// TwinCAT 3 PLC project CX_322E40
// libraries:
//   Tc2_ControllerToolbox, * (Beckhoff Automation GmbH)
//   Tc2_Coupler, * (Beckhoff Automation GmbH)
//   Tc2_DALI, * (Beckhoff Automation GmbH)
//   Tc2_EIB, * (Beckhoff Automation GmbH)
//   Tc2_EtherCAT, * (Beckhoff Automation GmbH)
//   Tc2_IoFunctions, * (Beckhoff Automation GmbH)
//   Tc2_LON, * (Beckhoff Automation GmbH)
//   Tc2_MBus, * (Beckhoff Automation GmbH)
//   Tc2_ModbusRTU, * (Beckhoff Automation GmbH)
//   Tc2_ModbusSrv, * (Beckhoff Automation GmbH)
//   Tc2_Standard, * (Beckhoff Automation GmbH)
//   Tc2_Standard, * (Beckhoff Automation GmbH)
//   Tc2_System, * (Beckhoff Automation GmbH)
//   Tc2_System, * (Beckhoff Automation GmbH)
//   Tc2_SystemCX, * (Beckhoff Automation GmbH)
//   Tc2_Utilities, * (Beckhoff Automation GmbH)
//   Tc3_Module, * (Beckhoff Automation GmbH)
//   Tc3_Module, * (Beckhoff Automation GmbH)
//   Tc3_PLCopen_OpcUa, * (Beckhoff Automation GmbH)
// project tree:
//   / ComTask.TcTTO, MBus_Zaehler_Task.TcTTO (not stored), Standard.TcTTO (not stored)
//   Data types/Anlagen/M2M/ WZM_EMAG_VLC100Y.TcDUT (not stored) (excluded from build)
//   Data types/Anlagen/ Machine2Machine.TcDUT (not stored)
//   Data types/Einzelanlagen/Absorptionskältemaschine %28AKM%29/ ST_AKM_Parameter.TcDUT (not stored), ST_AKM_Steuerung.TcDUT (not stored), ST_AKM_Zustand.TcDUT (not stored)
//   Data types/Einzelanlagen/Ampel/ ST_Ampel_Parameter.TcDUT (not stored), ST_Ampel_Steuerung.TcDUT, ST_Ampel_Zustand.TcDUT (not stored)
//   Data types/Einzelanlagen/Beleuchtung %28Bel%29/ ST_Bel_Lampen_Monitoring.TcDUT (not stored), ST_Bel_Parameter.TcDUT (not stored), ST_Bel_RGBW_Steuerung.TcDUT (not stored), ST_Bel_RGBW_Zustand.TcDUT (not stored), ST_Bel_Stellwert.TcDUT (not stored), ST_Bel_Steuerung.TcDUT (not stored), ST_Bel_Zustand.TcDUT (not stored)
//   Data types/Einzelanlagen/Betonspeicher %28BSp%29/ ST_BSp_Parameter.TcDUT (not stored), ST_Bsp_Steuerung.TcDUT (not stored), ST_BSp_Zustand.TcDUT (not stored)
//   Data types/Einzelanlagen/Blockheizkraftwerk %28BHKW%29/ ST_BHKW_Parameter.TcDUT (not stored), ST_BHKW_Stellwert.TcDUT (not stored), ST_BHKW_Steuerung.TcDUT (not stored), ST_BHKW_Zustand.TcDUT (not stored)
//   Data types/Einzelanlagen/Brennwertkessel %28BWK%29/ ST_BWK_Parameter.TcDUT (not stored), ST_BWK_Stellwert.TcDUT (not stored), ST_BWK_Steuerung.TcDUT (not stored), ST_BWK_Zustand.TcDUT (not stored)
//   Data types/Einzelanlagen/DC Schaltschrank %28DCSS%29/ ST_DCSS_Zustand.TcDUT (not stored)
//   Data types/Einzelanlagen/Druckluftkompressor %28DLK%29/ ST_DLK_Parameter.TcDUT (not stored), ST_DLK_Zustand.TcDUT (not stored)
//   Data types/Einzelanlagen/Drucksensor %28DS%29/ ST_DS_Parameter.TcDUT (not stored), ST_DS_Zustand.TcDUT (not stored)
//   Data types/Einzelanlagen/Fenster/ ST_Fenster_Parameter.TcDUT (not stored), ST_Fenster_Stellwert.TcDUT, ST_Fenster_Steuerung.TcDUT (not stored), ST_Fenster_Zustand.TcDUT (not stored)
//   Data types/Einzelanlagen/Gaszaehler %28GZ%29/ ST_GZ_DLK_Zustand.TcDUT (not stored), ST_GZ_Zustand.TcDUT (not stored)
//   Data types/Einzelanlagen/Haerteofen %28HO%29/ ST_HO_Parameter.TcDUT (not stored), ST_HO_Zustand.TcDUT (not stored)
//   Data types/Einzelanlagen/Heizstaebe %28HS%29/ ST_HS_Zustand.TcDUT (not stored)
//   Data types/Einzelanlagen/Hybrider Energiespeicher %28HES%29/ ST_HES_Parameter.TcDUT (not stored), ST_HES_Zustand.TcDUT (not stored)
//   Data types/Einzelanlagen/Kaeltekompressor %28KK%29/ ST_KKKW_Zustand.TcDUT (not stored)
//   Data types/Einzelanlagen/Lueftungsanlage %28LA%29/ ST_LA_Parameter.TcDUT (not stored), ST_LA_Stellwert.TcDUT (not stored), ST_LA_Steuerung.TcDUT (not stored), ST_LA_Zustand.TcDUT (not stored)
//   Data types/Einzelanlagen/Maschinenversorgung %28MV%29/ ST_MV_EMAG_VLC100Y_Zustand.TcDUT (not stored), ST_MV_HD_Zustand.TcDUT (not stored), ST_MV_JAVA_Parameter.TcDUT (not stored), ST_MV_JAVA_Zustand.TcDUT (not stored), ST_MV_MAFAC_GT_Parameter.TcDUT (not stored), ST_MV_MAFAC_GT_Zustand.TcDUT (not stored)
//   Data types/Einzelanlagen/Pufferspeicher %28PSp%29/ ST_PSp_Parameter.TcDUT (not stored), ST_PSp_Zustand.TcDUT (not stored)
//   Data types/Einzelanlagen/Pumpe %28Pu%29/ ST_PU_Genibus.TcDUT (not stored), ST_PU_Parameter.TcDUT (not stored), ST_PU_Stellwert.TcDUT (not stored), ST_PU_Steuerung.TcDUT (not stored), ST_PU_Zustand.TcDUT (not stored)
//   Data types/Einzelanlagen/Pumpe_lesend %28PU_Les%29/ ST_PU_les_Zustand.TcDUT (not stored)
//   Data types/Einzelanlagen/Pumpe_Schuetz %28PU_Schuetz%29/ ST_PU_Schuetz_Parameter.TcDUT (not stored), ST_PU_Schuetz_Stellwert.TcDUT (not stored), ST_PU_Schuetz_Steuerung.TcDUT (not stored), ST_PU_Schuetz_Zustand.TcDUT (not stored)
//   Data types/Einzelanlagen/Regelventil %28RV%29/ ST_RV_Parameter.TcDUT (not stored), ST_RV_Stellwert.TcDUT (not stored), ST_RV_Steuerung.TcDUT (not stored), ST_RV_Zustand.TcDUT (not stored)
//   Data types/Einzelanlagen/Regelventil_lesend %28RV_les%29/ ST_RV_les_Stellwert.TcDUT (not stored), ST_RV_les_Zustand.TcDUT (not stored)
//   Data types/Einzelanlagen/RGBW-Kanal/ ST_RGBW_Steuerung.TcDUT, ST_RGBW_Zustand.TcDUT (not stored)
//   Data types/Einzelanlagen/Signallampe GLT %28SL%29/ ST_SL_Parameter.TcDUT (not stored), ST_SL_Stellwert.TcDUT (not stored), ST_SL_Steuerung.TcDUT (not stored), ST_SL_Zustand.TcDUT (not stored)
//   Data types/Einzelanlagen/Stellventil %28SV%29 _ mit Status %28SVs%29/ ST_SVs_504_505_Zustand.TcDUT (not stored), ST_SVs_Zustand.TcDUT (not stored), ST_SV_Parameter.TcDUT (not stored), ST_SV_Stellwert.TcDUT (not stored), ST_SV_Steuerung.TcDUT (not stored), ST_SV_Zustand.TcDUT (not stored)
//   Data types/Einzelanlagen/Stromzaehler %28SZ%29/ ST_NSHV_Zustand.TcDUT (not stored), ST_SZ_Zustand.TcDUT (not stored)
//   Data types/Einzelanlagen/Tempfuehler%28TF%29/ ST_System_TF_Zustand.TcDUT (not stored)
//   Data types/Einzelanlagen/Waermepumpe %28WP%29/ ST_WP_Parameter.TcDUT (not stored), ST_WP_Stellwert.TcDUT (not stored), ST_WP_Steuerung.TcDUT (not stored), ST_WP_Zustand.TcDUT (not stored)
//   Data types/Einzelanlagen/Waermezaehler %28WZ%29/ ST_WZ_Zustand.TcDUT (not stored)
//   Data types/Library/Allgemein/ ST_Steuerung_auto_manu_BOOL.TcDUT (not stored), ST_Steuerung_auto_manu_opti_BOOL.TcDUT (not stored), ST_Steuerung_auto_manu_opti_REAL.TcDUT (not stored), ST_Steuerung_auto_manu_opti_SINT.TcDUT, ST_Steuerung_auto_manu_String.TcDUT, ST_Zustand_Netze_Anford.TcDUT (not stored), ST_Zustand_Netz_Anford.TcDUT (not stored)
//   Data types/Library/Bus_Systeme/ PB_64Byte.TcDUT (not stored), PB_Anfrage.TcDUT, PB_Dateneintrag.TcDUT, PB_GenibusType.TcDUT (not stored), PB_UMG604.TcDUT, ST_NSHV_Modbus.TcDUT
//   Data types/Management/ ST_FB_MGMT_Parameter.TcDUT (not stored), ST_FB_MGMT_Stellwert.TcDUT (not stored), ST_FB_MGMT_Steuerung.TcDUT, ST_FB_MGMT_Zustand.TcDUT (not stored), ST_MGMT_ThNTZ_Aktor_Parameter.TcDUT, ST_MGMT_ThNTZ_Aktor_Stellwert.TcDUT (not stored), ST_MGMT_ThNTZ_Aktor_Zustand.TcDUT (not stored)
//   Data types/Netze/ ST_Netze_Parameter.TcDUT (not stored), ST_Parameter_NTZ_Aktor_Regelung.TcDUT (not stored), ST_ThNTZ_Aktor.TcDUT, ST_ThNTZ_Parameter.TcDUT, ST_ThNTZ_Stellwert.TcDUT, ST_ThNTZ_Steuerung.TcDUT (not stored), ST_ThNTZ_Zustand.TcDUT
//   Data types/OPC-UA/ OPC_UA_BOOL.TcDUT (not stored), OPC_UA_REAL.TcDUT (not stored), ST_OPCUA_Node_BOOL.TcDUT, ST_OPCUA_Node_REAL.TcDUT (not stored), ST_OPCUA_Server.TcDUT, ST_OPC_UA_Node.TcDUT
//   Data types/Sonstige/ ST_GA_global.TcDUT (not stored), ST_Initialisierungsroutine.TcDUT (not stored)
//   Data types/Systeme/Anlagenversorgung %28AV%29/System Druckluftkompressor %28DLK%29/ ST_System_DLK_Parameter.TcDUT (not stored), ST_System_DLK_Stellwert.TcDUT (not stored), ST_System_DLK_Steuerung.TcDUT (not stored), ST_System_DLK_Zustand.TcDUT (not stored)
//   Data types/Systeme/Anlagenversorgung %28AV%29/System HybriderEnergiespeicher %28HES%29/ ST_System_HES_Parameter.TcDUT (not stored), ST_System_HES_Stellwert.TcDUT (not stored), ST_System_HES_Steuerung.TcDUT (not stored), ST_System_HES_Zustand.TcDUT (not stored)
//   Data types/Systeme/Anlagenversorgung %28AV%29/System Härteofen %28HO%29/System Härteofen Heisswasser %28HOHW%29/ ST_System_HOHW_Parameter.TcDUT (not stored), ST_System_HOHW_Stellwert.TcDUT (not stored), ST_System_HOHW_Steuerung.TcDUT (not stored), ST_System_HOHW_Zustand.TcDUT (not stored)
//   Data types/Systeme/Anlagenversorgung %28AV%29/System Härteofen %28HO%29/System Härteofen Warmwasser %28HOWW%29/ ST_System_HOWW_Parameter.TcDUT (not stored), ST_System_HOWW_Stellwert.TcDUT (not stored), ST_System_HOWW_Steuerung.TcDUT (not stored), ST_System_HOWW_Zustand.TcDUT (not stored)
//   Data types/Systeme/Anlagenversorgung %28AV%29/System Maschinenversorgung Heisswasser %28MVHW%29/ ST_System_MVHW_Parameter.TcDUT (not stored), ST_System_MVHW_Stellwert.TcDUT (not stored), ST_System_MVHW_Steuerung.TcDUT (not stored), ST_System_MVHW_Zustand.TcDUT (not stored)
//   Data types/Systeme/Anlagenversorgung %28AV%29/System Maschinenversorgung Kaltwasser %28MVKW%29/ ST_System_MVKW_Parameter.TcDUT (not stored), ST_System_MVKW_Stellwert.TcDUT (not stored), ST_System_MVKW_Steuerung.TcDUT (not stored), ST_System_MVKW_Zustand.TcDUT (not stored)
//   Data types/Systeme/Anlagenversorgung %28AV%29/System Maschinenversorgung Warmwasser %28MVWW%29/ ST_System_MVWW_Parameter.TcDUT (not stored), ST_System_MVWW_Stellwert.TcDUT (not stored), ST_System_MVWW_Steuerung.TcDUT (not stored), ST_System_MVWW_Zustand.TcDUT (not stored)
//   Data types/Systeme/Beleuchtung %28Bel%29/ ST_System_Bel_Parameter.TcDUT (not stored), ST_System_Bel_Stellwert.TcDUT (not stored), ST_System_Bel_Steuerung.TcDUT (not stored), ST_System_Bel_Zustand.TcDUT (not stored)
//   Data types/Systeme/Heizung_Klima_Lueftung/Klima/ ST_Klima_Aussen.TcDUT (not stored), ST_Klima_Bueros.TcDUT (not stored), ST_Klima_Halle.TcDUT
//   Data types/Systeme/Heizung_Klima_Lueftung/Lueftungsanlage %28LA%29/ ST_System_LA_Parameter.TcDUT (not stored), ST_System_LA_Stellwert.TcDUT (not stored), ST_System_LA_Steuerung.TcDUT (not stored), ST_System_LA_Zustand.TcDUT (not stored)
//   Data types/Systeme/Heizung_Klima_Lueftung/Lueftungsanlage %28LA%29/System_Fenster/ ST_System_Fenster_Parameter.TcDUT (not stored), ST_System_Fenster_Stellwert.TcDUT (not stored), ST_System_Fenster_Steuerung.TcDUT (not stored), ST_System_Fenster_Zustand.TcDUT (not stored)
//   Data types/Systeme/Heizung_Klima_Lueftung/Statische Heizung %28SHZ%29/ ST_System_SHZ_Parameter.TcDUT (not stored), ST_System_SHZ_Stellwert.TcDUT (not stored), ST_System_SHZ_Steuerung.TcDUT (not stored), ST_System_SHZ_Zustand.TcDUT (not stored)
//   Data types/Systeme/Heizung_Klima_Lueftung/ ST_Parameter_Kennlinie_Heizung_Kuehlung.TcDUT, ST_Parameter_Nachtabsenkung.TcDUT (not stored)
//   Data types/Systeme/Heizung_Klima_Lueftung/System Fussbodentemperierung %28FBT%29/ ST_System_FBT_Parameter.TcDUT (not stored), ST_System_FBT_Stellwert.TcDUT (not stored), ST_System_FBT_Steuerung.TcDUT (not stored), ST_System_FBT_Zustand.TcDUT (not stored)
//   Data types/Systeme/Heizung_Klima_Lueftung/Wand- & Deckentemperierung %28WDT%29/ ST_System_WDT_Parameter.TcDUT (not stored), ST_System_WDT_Stellwert.TcDUT (not stored), ST_System_WDT_Steuerung.TcDUT (not stored), ST_System_WDT_Zustand.TcDUT (not stored)
//   Data types/Systeme/Kaeltekompressor/Kaeltekompressor Kaltwasser/ ST_System_KKKW_Parameter.TcDUT, ST_System_KKKW_Stellwert.TcDUT, ST_System_KKKW_Steuerung.TcDUT (not stored), ST_System_KKKW_Zustand.TcDUT
//   Data types/Systeme/Speicher/Betonspeicher %28BSp%29/ ST_System_BSp_Parameter.TcDUT (not stored), ST_System_BSp_Stellwert.TcDUT (not stored), ST_System_BSp_Steuerung.TcDUT (not stored), ST_System_BSp_Zustand.TcDUT (not stored)
//   Data types/Systeme/Speicher/Betonspeicher Kühlwasser %28BSp_KueW%29/ ST_System_BSp_KueW_Parameter.TcDUT (not stored), ST_System_BSp_KueW_Stellwert.TcDUT (not stored), ST_System_BSp_KueW_Steuerung.TcDUT (not stored), ST_System_BSp_KueW_Zustand.TcDUT (not stored)
//   Data types/Systeme/Speicher/Betonspeicher Verbindung %28BSp_Verb%29/ ST_System_BSp_Verb_Parameter.TcDUT (not stored), ST_System_BSp_Verb_Stellwert.TcDUT (not stored), ST_System_BSp_Verb_Steuerung.TcDUT (not stored), ST_System_BSp_Verb_Zustand.TcDUT (not stored)
//   Data types/Systeme/System_Ampel/ ST_Steuerung_auto_manu_opti_AMPELSIGNAL.TcDUT, ST_System_Ampel_Signal.TcDUT, ST_System_Ampel_Stellwert.TcDUT, ST_System_Ampel_Steuerung.TcDUT (not stored), ST_System_Ampel_Zustand.TcDUT
//   Data types/Systeme/Wandler/Aussenfassadenaktivierung %28AFA%29/ ST_System_AFA_Parameter.TcDUT (not stored), ST_System_AFA_Stellwert.TcDUT (not stored), ST_System_AFA_Steuerung.TcDUT (not stored), ST_System_AFA_Zustand.TcDUT (not stored)
//   Data types/Systeme/Wandler/System Absorptionskältemaschine %28AKM%29/ ST_System_AKM_Parameter.TcDUT (not stored), ST_System_AKM_Stellwert.TcDUT (not stored), ST_System_AKM_Steuerung.TcDUT (not stored), ST_System_AKM_Zustand.TcDUT (not stored)
//   Data types/Systeme/Wandler/System Blockheizkraftwerk %28BHKW%29/ ST_System_BHKW_Parameter.TcDUT (not stored), ST_System_BHKW_Stellwert.TcDUT (not stored), ST_System_BHKW_Steuerung.TcDUT (not stored), ST_System_BHKW_Zustand.TcDUT (not stored)
//   Data types/Systeme/Wandler/System Brennwertkessel %28BWK%29/ ST_System_BWK_Parameter.TcDUT (not stored), ST_System_BWK_Stellwert.TcDUT (not stored), ST_System_BWK_Steuerung.TcDUT (not stored), ST_System_BWK_Zustand.TcDUT (not stored)
//   Data types/Systeme/Wandler/System Heizstaebe %28HS%29/ ST_System_HS_Parameter.TcDUT (not stored), ST_System_HS_Stellwert.TcDUT (not stored), ST_System_HS_Steuerung.TcDUT (not stored), ST_System_HS_Zustand.TcDUT (not stored)
//   Data types/Systeme/Wandler/System Waermepumpe %28WP%29/ ST_System_WP_Parameter.TcDUT (not stored), ST_System_WP_Stellwert.TcDUT (not stored), ST_System_WP_Steuerung.TcDUT (not stored), ST_System_WP_Zustand.TcDUT (not stored)
//   Data types/Systeme/Wandler/System Wärmetauscher Warm-Heisswasser %28WT_WHW%29/ ST_System_WT_HWW_Parameter.TcDUT (not stored), ST_System_WT_HWW_Stellwert.TcDUT (not stored), ST_System_WT_HWW_Steuerung.TcDUT (not stored), ST_System_WT_HWW_Zustand.TcDUT (not stored)
//   Global Variables/Anlagen Variablen/ Con_AFA.TcGVL, Con_AKM.TcGVL (not stored), Con_Bel.TcGVL (not stored), Con_BHKW.TcGVL, Con_BSp.TcGVL, Con_BWK.TcGVL (not stored), Con_DLK.TcGVL (not stored), Con_FBT.TcGVL (not stored), Con_HO.TcGVL, Con_HS.TcGVL (not stored), Con_KKKW.TcGVL, Con_MGMT.TcGVL (not stored), Con_MVKW.TcGVL (not stored), Con_MVWW.TcGVL, Con_PU.TcGVL, Con_RV.TcGVL (not stored), Con_SHZ.TcGVL, Con_SV.TcGVL, Con_ThNTZ.TcGVL, Con_WDT.TcGVL, Con_WP.TcGVL (not stored), Con_WT.TcGVL (not stored)
//   Global Variables/Bus_Systeme/ Modbus.TcGVL (not stored), M_Bus.TcGVL, Profibus.TcGVL
//   Global Variables/ Globale_Variablen.TcGVL (not stored), Global_Checks.TcGVL (not stored), Global_Variables.TcGVL, Variablen_Konfiguration.TcGVL (not stored)
//   POUs/Checks/ CheckBounds.TcPOU, CheckDivByte.TcPOU (not stored), CheckDivDint.TcPOU (not stored), CheckDivDWord.TcPOU, CheckDivInt.TcPOU (not stored), CheckDivLreal.TcPOU (not stored), CheckDivReal.TcPOU, CheckDivSInt.TcPOU (not stored), CheckDivWord.TcPOU, CheckRangeSigned.TcPOU (not stored), CheckRangeUnsigned.TcPOU
//   POUs/ com_task.TcPOU, Error_Catch.TcPOU, FB_GA_Allgemein.TcPOU (not stored), FB_Initialisierungsroutine.TcPOU, MAIN.TcPOU (not stored), MBUS_WZaehler.TcPOU, MBUS_Zaehler.TcPOU (not stored), P_EIB.TcPOU (excluded from build)
//   POUs/Einzelanlagen/Absorptionskältemaschine %28AKM%29/ FB_AKM.TcPOU (not stored), FB_AKM_Zuweisung.TcPOU (not stored)
//   POUs/Einzelanlagen/Ampel/ FB_Ampel.TcPOU (not stored), FB_Ampel_Out.TcPOU
//   POUs/Einzelanlagen/Beleuchtung %28Bel%29/Bel_RGBW/ FB_Bel_Einzel_farbe.TcPOU (not stored), FB_Bel_Einzel_farbe_1.TcPOU (not stored), FB_Bel_RGBW.TcPOU (not stored), FB_Bel_RGBW_Ablaufsteuerung.TcPOU (not stored), FB_Bel_RGBW_Logik.TcPOU (not stored), FB_Bel_RGBW_Regelung.TcPOU (not stored), FB_Bel_RGBW_Sued.TcPOU (not stored) (excluded from build)
//   POUs/Einzelanlagen/Beleuchtung %28Bel%29/ FB_Bel.TcPOU (not stored), FB_Bel_Ablaufsteuerung.TcPOU (not stored), FB_Bel_Filter.TcPOU (not stored), FB_Bel_Input.TcPOU (not stored), FB_Bel_Lichtsensor.TcPOU (not stored), FB_Bel_Logik.TcPOU (not stored), FB_Bel_Monitoring.TcPOU (not stored), FB_Bel_Output.TcPOU (not stored), FB_Bel_Sollwertscheck.TcPOU (not stored), FB_Bel_Stellwertscheck.TcPOU (not stored), FB_Bel_Steuerung.TcPOU (not stored), FB_Bel_Taster.TcPOU (not stored), FB_Bel_Taster_Steuerung.TcPOU (not stored), FB_Bel_Zustandscheck.TcPOU (not stored), F_Bel_Daten_Lesen.TcPOU (not stored), F_Bel_Daten_Schreiben.TcPOU (not stored)
//   POUs/Einzelanlagen/Betonspeicher %28BSp%29/ FB_BSp.TcPOU (not stored), FB_BSp_Input.TcPOU (not stored), FB_BSp_Zustandscheck.TcPOU (not stored)
//   POUs/Einzelanlagen/Blockheizkraftwerk %28BHKW%29/ FB_BHKW.TcPOU (not stored), FB_BHKW_Ablaufsteuerung.TcPOU (not stored), FB_BHKW_Input.TcPOU (not stored), FB_BHKW_Logik.TcPOU (not stored), FB_BHKW_Modbus.TcPOU (not stored), FB_BHKW_Output.TcPOU (not stored), FB_BHKW_Regelung.TcPOU (not stored), FB_BHKW_Sollwertscheck.TcPOU (not stored), FB_BHKW_Stellwertscheck.TcPOU (not stored), FB_BHKW_Zustandscheck.TcPOU (not stored), F_BHKW_Daten_Schreiben.TcPOU (not stored)
//   POUs/Einzelanlagen/Brennwertkessel %28BWK%29/ FB_BWK.TcPOU (not stored), FB_BWK_Ablaufsteuerung.TcPOU (not stored), FB_BWK_Input.TcPOU (not stored), FB_BWK_Logik.TcPOU (not stored), FB_BWK_Output.TcPOU (not stored), FB_BWK_Regelung.TcPOU (not stored), FB_BWK_SchreibeDaten.TcPOU (not stored), FB_BWK_Sollwertscheck.TcPOU (not stored), FB_BWK_Stellwertscheck.TcPOU (not stored), FB_BWK_Zustandscheck.TcPOU (not stored), LON_COM.TcPOU (not stored), LON_IN_OUT.TcPOU (not stored)
//   POUs/Einzelanlagen/DC Schaltschrank %28DCSS%29/ FB_DCSS.TcPOU (not stored)
//   POUs/Einzelanlagen/Druckluftkompressor %28DLK%29/ FB_DLK.TcPOU (not stored), FB_DLK_INIt.TcPOU (not stored), FB_DLK_Input.TcPOU (not stored), FB_DLK_Zustandscheck.TcPOU (not stored)
//   POUs/Einzelanlagen/Drucksensor/ FB_DS.TcPOU, FB_DS_Input.TcPOU, FB_DS_Zustandscheck.TcPOU
//   POUs/Einzelanlagen/Fenster/ FB_Fenster.TcPOU (not stored), FB_Fenster_Ablaufsteuerung.TcPOU (not stored), FB_Fenster_Logik.TcPOU, FB_Fenster_Output.TcPOU (not stored), FB_Fenster_Zustandscheck.TcPOU (not stored), F_Fenster_Daten_Lesen.TcPOU (not stored)
//   POUs/Einzelanlagen/Gaszähler/ FB_Gaszaehler.TcPOU (not stored), FB_GZ_DLK.TcPOU (not stored)
//   POUs/Einzelanlagen/Haerteofen %28HO%29/ FB_HO.TcPOU (not stored)
//   POUs/Einzelanlagen/Heizstab %28HS%29/ FB_HS.TcPOU (not stored)
//   POUs/Einzelanlagen/Hybrider Energiespeicher %28HES%29/ FB_HES.TcPOU (not stored)
//   POUs/Einzelanlagen/Kaeltekompressor %28KK%29/Kaeltekompressor Kaltwasser %28KKKW%29/ FB_KKKW.TcPOU (not stored)
//   POUs/Einzelanlagen/Lueftungsanlage %28LA%29/ FB_LA.TcPOU (not stored), FB_LA_Zustandscheck.TcPOU (not stored)
//   POUs/Einzelanlagen/Maschinenversorgung %28MV%29/ FB_MV_EMAG_GT.TcPOU (not stored), FB_MV_EMAG_VLC100Y.TcPOU (not stored), FB_MV_HD.TcPOU (not stored), FB_MV_JAVA.TcPOU (not stored)
//   POUs/Einzelanlagen/Pufferspeicher %28PSp%29/ FB_PSp.TcPOU (not stored), FB_PSp_Input.TcPOU (not stored), FB_PSp_Zustandscheck.TcPOU (not stored)
//   POUs/Einzelanlagen/Pumpe %28PU%29/ FB_PU.TcPOU (not stored), FB_PU_Ablaufsteuerung.TcPOU (not stored), FB_PU_Genibus.TcPOU (not stored), FB_PU_Genibus_old.TcPOU (not stored), FB_PU_Input.TcPOU (not stored), FB_PU_Logik.TcPOU (not stored), FB_PU_Output.TcPOU (not stored), FB_PU_Regelung.TcPOU (not stored), FB_PU_Sollwertscheck.TcPOU (not stored), FB_PU_Zustandscheck.TcPOU (not stored), F_PU_Daten_Schreiben.TcPOU (not stored)
//   POUs/Einzelanlagen/Pumpe %28PU%29/PU_191/ FB_PU_191.TcPOU (not stored), FB_PU_191_Ablaufsteuerung.TcPOU (not stored), FB_PU_191_Input.TcPOU (not stored)
//   POUs/Einzelanlagen/Pumpe Status %28PU_St%29/ FB_PU_St.TcPOU (not stored), FB_PU_St_Zustandscheck.TcPOU (not stored)
//   POUs/Einzelanlagen/Pumpe_lesend %28PU_les%29/ FB_PU_les.TcPOU (not stored), FB_PU_les_Genibus.TcPOU (not stored), FB_PU_les_Input.TcPOU (not stored)
//   POUs/Einzelanlagen/Pumpe_Schuetz %28PU_Schuetz%29/ FB_PU_Schuetz.TcPOU (not stored), FB_PU_Schuetz_Ablaufsteuerung.TcPOU (not stored), FB_PU_Schuetz_Logik.TcPOU (not stored), FB_PU_Schuetz_Output.TcPOU (not stored), FB_PU_Schuetz_Zustandscheck.TcPOU (not stored), FB_PU_Stellwertscheck.TcPOU (not stored)
//   POUs/Einzelanlagen/Regelventil %28RV%29/ FB_RV.TcPOU (not stored), FB_RV_Ablaufsteuerung.TcPOU (not stored), FB_RV_Logik.TcPOU (not stored), FB_RV_Output.TcPOU (not stored), FB_RV_Regelung.TcPOU (not stored), FB_RV_Sollwertscheck.TcPOU (not stored), FB_RV_Stellwertscheck.TcPOU (not stored), FB_RV_Zustandscheck.TcPOU (not stored)
//   POUs/Einzelanlagen/Regelventil Status %28RV_St%29/ FB_RV_St.TcPOU (not stored), FB_RV_St_Zustandscheck.TcPOU (not stored)
//   POUs/Einzelanlagen/Regelventil_lesend %28RV_les%29/ FB_RV_les.TcPOU (not stored)
//   POUs/Einzelanlagen/RGBW-Kanal/ FB_RGBW.TcPOU (not stored), FB_RGBW_Zustandscheck.TcPOU
//   POUs/Einzelanlagen/Stellventil %28SV%29/ FB_SV.TcPOU (not stored), FB_SV_Ablaufsteuerung.TcPOU (not stored), FB_SV_Logik.TcPOU (not stored), FB_SV_Output.TcPOU (not stored), FB_SV_Zustandscheck.TcPOU (not stored), F_SV_Daten_Schreiben.TcPOU (not stored)
//   POUs/Einzelanlagen/Stellventil mit Status %28SVs%29/ FB_SVs.TcPOU (not stored), FB_SVs_Ablaufsteuerung.TcPOU (not stored), FB_SVs_Input.TcPOU (not stored), FB_SVs_Logik.TcPOU (not stored), FB_SVs_Output.TcPOU (not stored), FB_SVs_Zustandscheck.TcPOU (not stored)
//   POUs/Einzelanlagen/Stellventil mit Status %28SVs%29/FB_SVs_504_505/ FB_SVs_504_505.TcPOU (not stored), FB_SVs_504_505_Ablaufsteuerung.TcPOU (not stored), FB_SVs_504_505_Input.TcPOU (not stored), FB_SVs_504_505_Logik.TcPOU (not stored), FB_SVs_504_505_Zustandscheck.TcPOU (not stored)
//   POUs/Einzelanlagen/Stromzähler/ABB_Stromzaehler/ FB_ABB_Lesen.TcPOU, FB_Stromzaehler.TcPOU (not stored), FB_Stromzaehler_BHKW.TcPOU, FB_Stromzaehler_Gebaeude.TcPOU
//   POUs/Einzelanlagen/Stromzähler/Netzanschlusspunkt/ FB_NSHV_Wert_zuweisen.TcPOU (not stored), FB_Stromzaehler_NSHV_Modbus.TcPOU
//   POUs/Einzelanlagen/Tempfuehler/ FB_TF.TcPOU (not stored)
//   POUs/Einzelanlagen/Waermepumpe/ FB_WP.TcPOU (not stored), FB_WP_Ablaufsteuerung.TcPOU, FB_WP_Logik.TcPOU, FB_WP_SchreibeDaten.TcPOU, FB_WP_Zustandscheck.TcPOU
//   POUs/Einzelanlagen/Wetterstation/ FB_WS.TcPOU (not stored), FB_WS_Init.TcPOU (not stored), FB_WS_Input.TcPOU (not stored), FB_WS_Konvertierung.TcPOU, FB_WS_Konvertierung_OLD.TcPOU (not stored), FB_WS_Mittelung.TcPOU
//   POUs/Einzelanlagen/Wärmezähler/ FB_Waermezaehler_MollineC3.TcPOU, FB_Waermezaehler_WP.TcPOU
//   POUs/Initialisierung/ P_init_dauernd.TcPOU (not stored), P_Init_einmalig.TcPOU (not stored)
//   POUs/Kommunikation/ FB_BUFFER_INT_TO_REAL.TcPOU, FB_BUFFER_REAL_TO_REAL.TcPOU, FB_BUFFER_UDINT_TO_REAL.TcPOU, OPC_UA_READ.TcPOU (not stored), OPC_UA_WRITE.TcPOU (not stored)
//   POUs/Library %28allgemein%29/ FB_SetResetFallTrigger.TcPOU (not stored), IEEE32_TO_REAL.TcPOU (not stored)
//   POUs/Management/Alte Struktur/ FB_MGMT_ThNTZ.TcPOU, FB_MGMT_ThNTZ_Aktor.TcPOU
//   POUs/Management/ FB_MGMT.TcPOU, FB_MGMT_Ablaufsteuerung.TcPOU, FB_MGMT_BSp.TcPOU (not stored), FB_MGMT_Logik.TcPOU, FB_MGMT_Regelung.TcPOU, FB_MGMT_Sollwertscheck.TcPOU, FB_MGMT_Zustandscheck.TcPOU (not stored), FB_Zuweisungen.TcPOU
//   POUs/OPC_UA_Client_Maschienen %28Romtech _ alt%29/ AKM_941_Read_BOOL.TcPOU (not stored) (excluded from build), AKM_941_Read_REAL.TcPOU (not stored) (excluded from build), AKM_941_Write_BOOL.TcPOU (not stored) (excluded from build), AKM_941_Write_REAL.TcPOU (not stored) (excluded from build), IVA_Ofen_Read_BOOL.TcPOU (not stored), IVA_Ofen_Read_REAL.TcPOU (not stored), PRG_Read_LREAL.TcPOU (not stored), SMS_Speicher_Read_BOOL.TcPOU (not stored) (excluded from build), SMS_Speicher_Read_REAL.TcPOU (not stored) (excluded from build)
//   POUs/Systeme/Anlagenversorgung %28AV%29/ FB_AV.TcPOU (not stored)
//   POUs/Systeme/Anlagenversorgung %28AV%29/Kühlung Druckluftkompressor %28DLK%29/ FB_System_DLK_951.TcPOU (not stored), FB_System_DLK_Ablaufsteuerung.TcPOU (not stored), FB_System_DLK_Logik.TcPOU (not stored), FB_System_DLK_Stellwertscheck.TcPOU (not stored), FB_System_DLK_Zustandscheck.TcPOU (not stored)
//   POUs/Systeme/Anlagenversorgung %28AV%29/Kühlung Hybrider Energiespeicher %28HES%29/ FB_System_HES_991.TcPOU (not stored), FB_System_HES_Ablaufsteuerung.TcPOU (not stored), FB_System_HES_Logik.TcPOU (not stored), FB_System_HES_Zustandscheck.TcPOU (not stored)
//   POUs/Systeme/Anlagenversorgung %28AV%29/Maschinenversorgung Heisswasser %28MVHW%29/ FB_System_MVHW_300.TcPOU (not stored), FB_System_MVHW_Ablaufsteuerung.TcPOU (not stored), FB_System_MVHW_Logik.TcPOU (not stored), FB_System_MVHW_Zustandscheck.TcPOU (not stored)
//   POUs/Systeme/Anlagenversorgung %28AV%29/Maschinenversorgung Kaltwasser %28MVKW%29/ FB_System_MVKW_100.TcPOU (not stored), FB_System_MVKW_Ablaufsteuerung.TcPOU (not stored), FB_System_MVKW_Logik.TcPOU (not stored), FB_System_MVKW_Zustandscheck.TcPOU (not stored)
//   POUs/Systeme/Anlagenversorgung %28AV%29/Maschinenversorgung Warmwasser %28MVWW%29/ FB_System_MVWW_245.TcPOU (not stored), FB_System_MVWW_Ablaufsteuerung.TcPOU (not stored), FB_System_MVWW_Logik.TcPOU (not stored), FB_System_MVWW_Sollwertscheck.TcPOU (not stored), FB_System_MVWW_Stellwertscheck.TcPOU (not stored), FB_System_MVWW_Zustandscheck.TcPOU (not stored)
//   POUs/Systeme/Anlagenversorgung %28AV%29/System Härteofen %28HO%29/ FB_System_HO_961.TcPOU (not stored)
//   POUs/Systeme/Anlagenversorgung %28AV%29/System Härteofen %28HO%29/System Härteofen Heisswasser %28HOHW%29/ FB_System_HOHW_361.TcPOU (not stored), FB_System_HOHW_Ablaufsteuerung.TcPOU (not stored), FB_System_HOHW_Logik.TcPOU (not stored), FB_System_HOHW_Zustandscheck.TcPOU (not stored)
//   POUs/Systeme/Anlagenversorgung %28AV%29/System Härteofen %28HO%29/System Härteofen Warmwasser %28HOWW%29/ FB_System_HOWW_261.TcPOU (not stored), FB_System_HOWW_Ablaufsteuerung.TcPOU (not stored), FB_System_HOWW_Logik.TcPOU (not stored), FB_System_HOWW_Zustandscheck.TcPOU (not stored)
//   POUs/Systeme/Heizung Lüftung Klimatisierung %28HLK%29/ FB_HLK.TcPOU (not stored)
//   POUs/Systeme/Heizung Lüftung Klimatisierung %28HLK%29/Fußbodentemperierung %28FBT%29/ FB_System_FBT_425.TcPOU (not stored), FB_System_FBT_Ablaufsteuerung.TcPOU (not stored), FB_System_FBT_Logik.TcPOU (not stored), FB_System_FBT_Regelung.TcPOU (not stored), FB_System_FBT_Sollwertscheck.TcPOU (not stored), FB_System_FBT_Stellwertscheck.TcPOU (not stored), FB_System_FBT_Zustandscheck.TcPOU (not stored)
//   POUs/Systeme/Heizung Lüftung Klimatisierung %28HLK%29/Raumlufttechnik %28RLT%29/Fenster %28FS%29/ FB_Fenster_Input.TcPOU (not stored), FB_System_Fenster.TcPOU (not stored), FB_System_Fenster_Logik.TcPOU (not stored), FB_System_Fenster_Regelung.TcPOU (not stored)
//   POUs/Systeme/Heizung Lüftung Klimatisierung %28HLK%29/Raumlufttechnik %28RLT%29/Lüftungsanlage %28LA%29/ FB_System_LA_955.TcPOU (not stored), FB_System_LA_Zustandscheck.TcPOU (not stored), SETINBYTE.TcPOU (not stored)
//   POUs/Systeme/Heizung Lüftung Klimatisierung %28HLK%29/Statische Heizung %28SHZ%29/ FB_System_SHZ_350.TcPOU (not stored), FB_System_SHZ_Ablaufsteuerung.TcPOU (not stored), FB_System_SHZ_Logik.TcPOU (not stored), FB_System_SHZ_Regelung.TcPOU (not stored), FB_System_SHZ_Sollwertscheck.TcPOU (not stored), FB_System_SHZ_Stellwertscheck.TcPOU (not stored), FB_System_SHZ_Zustandscheck.TcPOU (not stored)
//   POUs/Systeme/Heizung Lüftung Klimatisierung %28HLK%29/Wand- & Deckentemperierung %28WDT%29/ FB_System_WDT_500.TcPOU (not stored), FB_System_WDT_Ablaufsteuerung.TcPOU (not stored), FB_System_WDT_Logik.TcPOU (not stored), FB_System_WDT_Regelung.TcPOU (not stored), FB_System_WDT_Sollwertscheck.TcPOU (not stored), FB_System_WDT_Stellwertscheck.TcPOU (not stored), FB_System_WDT_Zustandscheck.TcPOU (not stored)
//   POUs/Systeme/Netze %28NTZ%29/ FB_HW_Zuweisungen.TcPOU (not stored), FB_KW_Zuweisungen.TcPOU (not stored), FB_NTZ.TcPOU (not stored), FB_NTZ_HW.TcPOU (not stored), FB_NTZ_KW.TcPOU (not stored), FB_NTZ_WW.TcPOU (not stored), FB_ThNTZ_Ablaufsteuerung.TcPOU (not stored), FB_ThNTZ_Logik.TcPOU (not stored), FB_ThNTZ_Regelung_Heissnetz.TcPOU (not stored), FB_ThNTZ_Regelung_Kaltnetz.TcPOU (not stored), FB_ThNTZ_Regelung_Warmnetz.TcPOU (not stored), FB_ThNTZ_Sollwertscheck.TcPOU (not stored), FB_ThNTZ_Zustandscheck.TcPOU (not stored), FB_WW_Zuweisungen.TcPOU (not stored)
//   POUs/Systeme/Sonstiges/Beleuchtung/Beleuchtung Außen/ FB_System_BelAu.TcPOU, FB_System_BelAu_Ablaufsteuerung.TcPOU, FB_System_BelAu_Logik.TcPOU, FB_System_BelAu_Regelung.TcPOU (not stored), FB_System_BelAu_Sensorik.TcPOU (not stored), FB_System_BelAu_Sollwertscheck.TcPOU, FB_System_BelAu_Stellwertscheck.TcPOU (not stored), FB_System_BelAu_Zustandscheck.TcPOU (not stored)
//   POUs/Systeme/Sonstiges/Beleuchtung/Beleuchtung Halle/ FB_System_BelHa.TcPOU (not stored), FB_System_BelHa_Ablaufsteuerung.TcPOU (not stored), FB_System_BelHa_Logik.TcPOU, FB_System_BelHa_Regelung.TcPOU (not stored), FB_System_BelHa_Sensorik.TcPOU (not stored), FB_System_BelHa_Sollwertscheck.TcPOU, FB_System_BelHa_Stellwertscheck.TcPOU (not stored), FB_System_BelHa_Zustandscheck.TcPOU (not stored)
//   POUs/Systeme/Sonstiges/Beleuchtung/ FB_Beleuchtung.TcPOU (not stored), FB_System_Bel_Zustandscheck.TcPOU
//   POUs/Systeme/Sonstiges/Signal_Ampel/ FB_System_Ampel.TcPOU (not stored), FB_System_Ampel_Sollwertscheck.TcPOU (not stored)
//   POUs/Systeme/Speicher %28SPR%29/Betonspeicher %28BSp%29/ FB_System_BSp_795.TcPOU (not stored), FB_System_BSp_795_Zustandscheck.TcPOU (not stored), FB_System_BSp_797.TcPOU (not stored), FB_System_BSp_797_Zustandscheck.TcPOU (not stored), FB_System_BSp_Ablaufsteuerung.TcPOU (not stored), FB_System_BSp_Logik.TcPOU (not stored), FB_System_BSp_Regelung.TcPOU (not stored), FB_System_BSp_Sollwertscheck.TcPOU (not stored), FB_System_BSp_Stellwertscheck.TcPOU (not stored)
//   POUs/Systeme/Speicher %28SPR%29/ FB_SPR.TcPOU (not stored)
//   POUs/Systeme/Wandler %28WDL%29/Absorptionskältemaschine %28AKM%29/ FB_System_AKM_941.TcPOU (not stored), FB_System_AKM_Ablaufsteuerung.TcPOU (not stored), FB_System_AKM_Logik.TcPOU (not stored), FB_System_AKM_Regelung.TcPOU (not stored), FB_System_AKM_Sollwertscheck.TcPOU (not stored), FB_System_AKM_Stellwertscheck.TcPOU (not stored), FB_System_AKM_Zustandscheck.TcPOU (not stored), FB_ThNTZ_Stellwertscheck.TcPOU (not stored)
//   POUs/Systeme/Wandler %28WDL%29/Aussenfassadenaktivierung %28AFA%29/ FB_System_AFA_600.TcPOU (not stored), FB_System_AFA_Ablaufsteuerung.TcPOU (not stored), FB_System_AFA_Logik.TcPOU (not stored), FB_System_AFA_Regelung.TcPOU (not stored), FB_System_AFA_Sollwertscheck.TcPOU (not stored), FB_System_AFA_Stellwertscheck.TcPOU (not stored), FB_System_AFA_Zustandscheck.TcPOU (not stored)
//   POUs/Systeme/Wandler %28WDL%29/Blockheizkraftwerke %28BHKWs%29/ FB_System_BHKW_921.TcPOU (not stored), FB_System_BHKW_922.TcPOU (not stored), FB_System_BHKW_Ablaufsteuerung.TcPOU (not stored), FB_System_BHKW_Logik.TcPOU (not stored), FB_System_BHKW_Sollwertscheck.TcPOU (not stored), FB_System_BHKW_Zustandscheck.TcPOU (not stored)
//   POUs/Systeme/Wandler %28WDL%29/Brennwertkessel %28BWK%29/ FB_System_BWK_931.TcPOU (not stored), FB_System_BWK_Ablaufsteuerung.TcPOU (not stored), FB_System_BWK_Logik.TcPOU (not stored), FB_System_BWK_Sollwertscheck.TcPOU (not stored), FB_System_BWK_Zustandscheck.TcPOU (not stored)
//   POUs/Systeme/Wandler %28WDL%29/ FB_WDL.TcPOU (not stored)
//   POUs/Systeme/Wandler %28WDL%29/Heizstaebe %28HS%29/ FB_System_HS_131.TcPOU (not stored), FB_System_HS_231.TcPOU (not stored), FB_System_HS_Logik.TcPOU (not stored), FB_System_HS_Regelung.TcPOU (not stored), FB_System_HS_Sollwertscheck.TcPOU (not stored), FB_System_HS_Zustandscheck.TcPOU (not stored)
//   POUs/Systeme/Wandler %28WDL%29/System_Kaeltekompressoren %28KK%29/Kältekompressor Kaltwasser/ FB_System_KKKW_145.TcPOU (not stored), FB_System_KKKW_Ablaufsteuerung.TcPOU (not stored), FB_System_KKKW_Logik.TcPOU (not stored), FB_System_KKKW_Sollwertscheck.TcPOU (not stored), FB_System_KKKW_Stellwertscheck.TcPOU (not stored), FB_System_KKKW_Zustandscheck.TcPOU (not stored)
//   POUs/Systeme/Wandler %28WDL%29/Waermepumpe %28WP%29/ FB_System_WP_946.TcPOU (not stored), FB_System_WP_Ablaufsteuerung.TcPOU (not stored), FB_System_WP_Logik.TcPOU (not stored), FB_System_WP_Zustandscheck.TcPOU (not stored)
//   POUs/Systeme/Wandler %28WDL%29/Wärmetauscher %28WT%29/ FB_System_WT_HWW_915.TcPOU (not stored), FB_System_WT_HWW_Ablaufsteuerung.TcPOU (not stored), FB_System_WT_HWW_Logik.TcPOU (not stored), FB_System_WT_HWW_Sollwertscheck.TcPOU (not stored), FB_System_WT_HWW_Zustandscheck.TcPOU (not stored)
//   POUs/Systeme/Zaehler %28ZAE%29/ FB_ZAE.TcPOU (not stored)
//   POUs/Umwelt/ FB_UMWELT.TcPOU, FB_UWT.TcPOU (not stored), FB_UW_Temp_Mittelung.TcPOU (not stored)

CONFIGURATION CX_322E40
    RESOURCE PLC ON TwinCAT3
        TASK ComTask(INTERVAL := T#25000us, PRIORITY := 6);
        PROGRAM com_task WITH ComTask : com_task;
    END_RESOURCE
END_CONFIGURATION

// ---- Data types/Einzelanlagen/Ampel/ST_Ampel_Steuerung.TcDUT
TYPE ST_Ampel_Steuerung :
STRUCT
	Freigabe			: ST_Steuerung_auto_manu_BOOL;
	Quittierung			: BOOL;
END_STRUCT
END_TYPE

// ---- Data types/Einzelanlagen/Fenster/ST_Fenster_Stellwert.TcDUT
TYPE ST_Fenster_Stellwert :
STRUCT
	Freigabe		: BOOL;
	Stellung		: BOOL;

	Fenster_AUF		: BOOL;
	Fenster_ZU		: BOOL;




END_STRUCT
END_TYPE

// ---- Data types/Einzelanlagen/RGBW-Kanal/ST_RGBW_Steuerung.TcDUT
TYPE ST_RGBW_Steuerung :
STRUCT
	Betrieb			: BOOL;
	Farbcode	: STRING;
END_STRUCT
END_TYPE

// ---- Data types/Library/Allgemein/ST_Steuerung_auto_manu_opti_SINT.TcDUT
TYPE ST_Steuerung_auto_manu_opti_SINT :
STRUCT
	auto			: SINT;
	manu			: SINT;
	manu_Modus		: BOOL;
	opti			: SINT;
	opti_Modus		: BOOL;
END_STRUCT
END_TYPE

// ---- Data types/Library/Allgemein/ST_Steuerung_auto_manu_String.TcDUT
TYPE ST_Steuerung_auto_manu_String :
STRUCT
	auto			: STRING;
	manu			: STRING;
	manu_Modus		: BOOL;
END_STRUCT
END_TYPE

// ---- Data types/Library/Bus_Systeme/PB_Anfrage.TcDUT
TYPE PB_Anfrage :
STRUCT
	pAuslass 			: PB_Dateneintrag;

	tAuslass 				: PB_Dateneintrag;
	
	tDruckTau			: PB_Dateneintrag;
	
	tUmgebung			: PB_Dateneintrag;

	tAqEin				: PB_Dateneintrag;

	tAqAus				: PB_Dateneintrag;
	
	mechState			: PB_Dateneintrag;

	hBetrieb				: PB_Dateneintrag;

	hGeringeLast			: PB_Dateneintrag;

	vErzeugtesVolumen	: PB_Dateneintrag;
END_STRUCT
END_TYPE

// ---- Data types/Library/Bus_Systeme/PB_Dateneintrag.TcDUT
TYPE PB_Dateneintrag :
STRUCT
	CANAdress 	: BYTE;
	Parameter 	: UINT;	
	Value		: UINT;
	Status		: WORD;
END_STRUCT
END_TYPE

// ---- Data types/Library/Bus_Systeme/PB_UMG604.TcDUT
TYPE PB_UMG604 :
(*Struktur für das Universalmessgerät 604 (Janitza) *)
STRUCT
	ProfilNummer		: BYTE;
	Wirkleistung 		: REAL;
	Blindleistung		: REAL;
	Scheinleistung	: REAL;
	Wirkarbeit		: REAL;
	Blindarbeit		: REAL;
	Scheinarbeit		: REAL;
	DiZaehlstand		: REAL;
	DiZustand		: REAL;
	DiLeistungswert	: REAL;
	NichtBelegt1		: REAL;
	NichtBelegt2		: REAL;
	NichtBelegt3		: REAL;
	NichtBelegt4		: REAL;
	NichtBelegt5		: REAL;
	NichtBelegt6		: REAL;
	NichtBelegt7		: REAL;
	NichtBelegt8		: REAL;
	NichtBelegt9		: REAL;
	NichtBelegt10		: REAL;
	NichtBelegt11		: REAL;
	NichtBelegt12		: REAL;
	NichtBelegt13		: REAL;
	NichtBelegt14		: REAL;
	NichtBelegt15		: REAL;
	NichtBelegt16		: REAL;
	NichtBelegt17		: REAL;
	NichtBelegt18		: REAL;
	NichtBelegt19		: REAL;
	NichtBelegt20		: REAL;
	NichtBelegt21		: REAL;
	NichtBelegt22		: REAL;
END_STRUCT
END_TYPE

// ---- Data types/Library/Bus_Systeme/ST_NSHV_Modbus.TcDUT
TYPE ST_NSHV_Modbus :
STRUCT
	Modbus_Unit_Online	: BOOL; (*True = online, False = Offline*)
	Modbus_Adresse1  : ARRAY[16#1000..16#1568] OF DWORD;
END_STRUCT
END_TYPE

// ---- Data types/Management/ST_FB_MGMT_Steuerung.TcDUT
TYPE ST_FB_MGMT_Steuerung :
STRUCT
	Freigabe			         : ST_Steuerung_auto_manu_BOOL;
	Freigabe_Deakt		: ST_Steuerung_auto_manu_BOOL;
	Betrieb_Anford		: ST_Steuerung_auto_manu_opti_BOOL;

	Regelung_Modus		: ST_Steuerung_auto_manu_opti_SINT;
	Regelung_Sollw		: ST_Steuerung_auto_manu_opti_REAL;
	Regelung_Sollw_Max	: ST_Steuerung_auto_manu_opti_REAL;
	Regelung_Sollw_Min	: ST_Steuerung_auto_manu_opti_REAL;

	Quittierung			: BOOL;

END_STRUCT
END_TYPE

// ---- Data types/Management/ST_MGMT_ThNTZ_Aktor_Parameter.TcDUT
TYPE ST_MGMT_ThNTZ_Aktor_Parameter :
STRUCT
	Anford_Netz_KW			: ST_Zustand_Netz_Anford;
	Anford_Netz_WW			: ST_Zustand_Netz_Anford;
	Anford_Netz_HW			: ST_Zustand_Netz_Anford;
	Regelung_Netz_KW		: ST_Parameter_NTZ_Aktor_Regelung;	(* Aktiv: Bool, Grenzwert_Oben: REAL, Grenzwert_Unten: REAL, Prioritaet: SINT;*)
	Regelung_Netz_WW		: ST_Parameter_NTZ_Aktor_Regelung;
	Regelung_Netz_HW		: ST_Parameter_NTZ_Aktor_Regelung;

	Kennlinie_Tctr			: DINT := 5000;
END_STRUCT
END_TYPE

// ---- Data types/Netze/ST_ThNTZ_Aktor.TcDUT
TYPE ST_ThNTZ_Aktor :
STRUCT
	Verfuegbarkeit_Heizer		: BOOL;
	Verfuegbarkeit_Kuehler	: BOOL;
	Betrieb_Heizer_Anford		: BOOL;
	Betrieb_Kuehler_Anford	: BOOL;
END_STRUCT
END_TYPE

// ---- Data types/Netze/ST_ThNTZ_Parameter.TcDUT
TYPE ST_ThNTZ_Parameter :
STRUCT
	Temp_Max				: REAL;
	Temp_Min				: REAL;
	Regelung_PI_Oben_Kp	: REAL;
	Regelung_PI_Oben_Tn	: DINT;
	Regelung_PI_Oben_Tctr	: DINT;

	Regelung_Sollw_KRITIKAL_OBEN_TEMP    : REAL;
	Regelung_Sollw_KRITIKAL_UNTEN_TEMP   : REAL;
	Regelung_Sollw_Max    : REAL;
	Regelung_Sollw_Min    : REAL;
	Regelung_Sollw_Max_Min : REAL;


	Stellwert_Leistung_Max		: REAL;
	Stellwert_Leistung_Min		: REAL;

	AutoQuittierung			: BOOL;



END_STRUCT
END_TYPE

// ---- Data types/Netze/ST_ThNTZ_Stellwert.TcDUT
TYPE ST_ThNTZ_Stellwert :
STRUCT
	Betrieb		: BOOL;
	Leistung	: REAL;
END_STRUCT
END_TYPE

// ---- Data types/Netze/ST_ThNTZ_Zustand.TcDUT
TYPE ST_ThNTZ_Zustand :
STRUCT
	Betrieb_Anford			: BOOL;
	Betrieb_Soll			: BOOL;
	Betrieb					: BOOL;

	Regelung_Modus				: SINT;
	Regelung_Sollw_Widerspruch	: BOOL;
	Regelung_Sollw				: REAL;
	Regelung_Sollw_Max          : REAL;
	Regelung_Sollw_Min			: REAL;

	Regelung_Sollw_Anford		: REAL;
	Regelung_Sollw_Oben			: REAL;
	Regelung_Sollw_Oben_Max		: REAL;
	Regelung_Sollw_Oben_Min		: REAL;
	Regelung_Sollw_Unten		: REAL;
	Regelung_Sollw_Unten_Max	: REAL;
	Regelung_Sollw_Unten_Min	: REAL;
	Regelung_Stellw				: REAL;
	Regelung_Istw				: REAL;

	Temp_Max				: REAL;
	Temp_Oben				: REAL;
	Temp_Min				: REAL;
	Temp_Unten				: REAL;

	Freigabe				: BOOL;
	Freigabe_Deakt			: BOOL;
	Freigabe_Code			: WORD;

    Netze_Anford            : ARRAY [1..20] OF ST_Zustand_Netze_Anford;

	Stoerung				: BOOL;
	Stoerung_Code			: WORD;

	Warnung					: BOOL;
	Warnung_Code			: WORD;

	Status					: SINT;

	Quittierung				: BOOL;

END_STRUCT
END_TYPE

// ---- Data types/OPC-UA/ST_OPCUA_Node_BOOL.TcDUT
TYPE ST_OPCUA_Node_BOOL :
STRUCT
	NodeID				: ST_UANodeID;
	NodeHdl				: DWORD;
	SizeOfDataType		: UDINT;
	NodeAddInfo			: ST_UANodeAdditionalInfo;
	TargetVar			: POINTER TO BOOL;
END_STRUCT
END_TYPE

// ---- Data types/OPC-UA/ST_OPCUA_Server.TcDUT
TYPE ST_OPCUA_Server :
STRUCT
	sServerURL				: STRING;
	SessionConnectInfo		: ST_UASessionConnectInfo := (	tConnectTimeout			:= T#5S,
															tSessionTimeout 		:= T#1M,
															sApplicationName		:= '',
															eSecurityMode 			:= eUASecurityMsgMode_None,
															eSecurityPolicyUri	 	:= eUASecurityPolicy_None,
															eTransportProfileUri 	:= eUATransportProfileUri_UATcp);
	tTimeout            	: TIME := T#5M;
	nConnectionHdl			: DWORD;
END_STRUCT
END_TYPE

// ---- Data types/OPC-UA/ST_OPC_UA_Node.TcDUT
TYPE ST_OPC_UA_Node :
STRUCT
	NodeID				: ST_UANodeID;
	NodeHdl				: DWORD;
	SizeOfDataType		: UDINT;
	NodeAddInfo			: ST_UANodeAdditionalInfo;
	TargetVar			: POINTER TO BOOL;
END_STRUCT
END_TYPE

// ---- Data types/Systeme/Heizung_Klima_Lueftung/Klima/ST_Klima_Halle.TcDUT
TYPE ST_Klima_Halle :
STRUCT
	Temperatur_Sektor1	: REAL;
	Temperatur_Sektor2	: REAL;
	Temperatur_Sektor3	: REAL;
END_STRUCT
END_TYPE

// ---- Data types/Systeme/Heizung_Klima_Lueftung/ST_Parameter_Kennlinie_Heizung_Kuehlung.TcDUT
TYPE ST_Parameter_Kennlinie_Heizung_Kuehlung :
STRUCT
	Temp_Vorl_Max			: REAL;
	Temp_Vorl_Min			: REAL;
	Temp_Aussen_Max			: REAL;
	Temp_Aussen_Min			: REAL;



END_STRUCT
END_TYPE

// ---- Data types/Systeme/Kaeltekompressor/Kaeltekompressor Kaltwasser/ST_System_KKKW_Parameter.TcDUT
TYPE ST_System_KKKW_Parameter :
STRUCT
		AutoQuittierung			: BOOL;
END_STRUCT
END_TYPE

// ---- Data types/Systeme/Kaeltekompressor/Kaeltekompressor Kaltwasser/ST_System_KKKW_Stellwert.TcDUT
TYPE ST_System_KKKW_Stellwert :
STRUCT
	Anford_Stellventil		: BOOL;
	Anford_Pumpe			: BOOL;
	Einschaltperiode_Max	: TIME := T#5S;
	Einschalten				: BOOL;
	Modus_Pumpe				: SINT;
	Sollw_Pumpe				: REAL;
END_STRUCT
END_TYPE

// ---- Data types/Systeme/Kaeltekompressor/Kaeltekompressor Kaltwasser/ST_System_KKKW_Zustand.TcDUT
TYPE ST_System_KKKW_Zustand :
STRUCT
	Betrieb_Anford			: BOOL;
	Betrieb_Soll				: BOOL;
	Betrieb					: BOOL;

	Regelung_Sollw			: REAL;
	Regelung_Modus				: SINT;

	Freigabe					: BOOL;
	Freigabe_Deakt			: BOOL;
	Freigabe_Code			: WORD;

	Stoerung					: BOOL;
	Stoerung_Code			: WORD;

	Warnung					: BOOL;
	Warnung_Code			: WORD;

	Status					: SINT;
	Status_Vorl				: BOOL;
	Status_Nachl				: BOOL;

	Status_Vorl_Stellventil	: BOOL;
	Status_Vorl_Pumpen		: BOOL;
	Status_Nachl_Stellventil: BOOL;
	Status_Nachl_Pumpen		: BOOL;
	Status_Wiedereinschalten: BOOL;

	Quittierung				: BOOL;

END_STRUCT
END_TYPE

// ---- Data types/Systeme/System_Ampel/ST_Steuerung_auto_manu_opti_AMPELSIGNAL.TcDUT
TYPE ST_Steuerung_auto_manu_opti_AMPELSIGNAL :
STRUCT
	auto			: ST_System_Ampel_Signal;
	manu			: ST_System_Ampel_Signal;
	manu_Modus		: BOOL;
	opti			: ST_System_Ampel_Signal;
	opti_Modus		: BOOL;
END_STRUCT
END_TYPE

// ---- Data types/Systeme/System_Ampel/ST_System_Ampel_Signal.TcDUT
TYPE ST_System_Ampel_Signal :
STRUCT
	Stellung_Rot		: BOOL;
	Stellung_Orange		: BOOL;
	Stellung_Gruen		: BOOL;
	Stellung_Blau		: BOOL;
	Stellung_Buzz		: BOOL;
END_STRUCT
END_TYPE

// ---- Data types/Systeme/System_Ampel/ST_System_Ampel_Stellwert.TcDUT
TYPE ST_System_Ampel_Stellwert :
STRUCT
	Stellung_Rot		: BOOL;
	Stellung_Orange		: BOOL;
	Stellung_Gruen		: BOOL;
	Stellung_Blau		: BOOL;
	Stellung_Buzz		: BOOL;
END_STRUCT
END_TYPE

// ---- Data types/Systeme/System_Ampel/ST_System_Ampel_Zustand.TcDUT
TYPE ST_System_Ampel_Zustand :
STRUCT
	Regelung_Sollw			: ST_System_Ampel_Signal;

	In_Ordnung			: BOOL;

	Stellung : ST_System_Ampel_Signal;
END_STRUCT
END_TYPE

// ---- Global Variables/Anlagen Variablen/Con_AFA.TcGVL
{attribute 'Tc2GvlVarNames'}
VAR_GLOBAL CONSTANT
	(* System_AFA_Zustand_Status *)
	E_System_AFA_Zustand_Status_Idle_Sperre			: SINT := 0;
	E_System_AFA_Zustand_Status_Betriebsbereit		: SINT := 1;
	E_System_AFA_Zustand_Status_Nachl_Pumpe			: SINT := 2;
	E_System_AFA_Zustand_Status_Vorl_Pumpe			: SINT := 3;
	E_System_AFA_Zustand_Status_Nachl_Regelventil	: SINT := 4;
	E_System_AFA_Zustand_Status_Vorl_Regelventil	: SINT := 5;
	E_System_AFA_Zustand_Status_Betrieb				: SINT := 6;
	E_System_AFA_Zustand_Status_Betrieb_Sperre		: SINT := 7;
	E_System_AFA_Zustand_Status_Stoerung			: SINT := 99;

	(* System_AFA_Zustand_Regelung_Modus *)
	E_System_AFA_Regelung_Modus_Wanddeckentemperierung		: SINT := -4;
	E_System_AFA_Regelung_Modus_Netz						: SINT := -5;

	E_System_AFA_Regelung_Modus_Waermeabsorber_Automatik	: SINT := 1;
	E_System_AFA_Regelung_Modus_Waermeabsorber_DachWaende	: SINT := 2;
	E_System_AFA_Regelung_Modus_Waermeabsorber_Dach			: SINT := 3;
	E_System_AFA_Regelung_Modus_Rueckkuehler_Automatik		: SINT := -1;
	E_System_AFA_Regelung_Modus_Rueckkuehler_DachWaende		: SINT := -2;
	E_System_AFA_Regelung_Modus_Rueckkuehler_Dach			: SINT := -3;

END_VAR

// ---- Global Variables/Anlagen Variablen/Con_BHKW.TcGVL
{attribute 'Tc2GvlVarNames'}
VAR_GLOBAL CONSTANT
	(* BHKW_Zustand_Status *)
	E_BHKW_Zustand_Status_Idle_Sperre			: SINT := 0;
	E_BHKW_Zustand_Status_Betriebsbereit		: SINT := 1;
	E_BHKW_Zustand_Status_Nachl					: SINT := 2;
	E_BHKW_Zustand_Status_Vorl					: SINT := 3;
	E_BHKW_Zustand_Status_Betrieb				: SINT := 4;
	E_BHKW_Zustand_Status_Betrieb_Sperre		: SINT := 5;
	E_BHKW_Zustand_Status_Stoerung				: SINT := 99;

	(* BHKW_Zustand_Regelung_Modus *)
	E_BHKW_Regelung_Modus_P						: SINT := 0;
	E_BHKW_Regelung_Modus_T_SH_Max				: SINT := 1;

	(* System_BHKW_Zustand_Status *)
	E_System_BHKW_Zustand_Status_Idle_Sperre		: SINT := 0;
	E_System_BHKW_Zustand_Status_Betriebsbereit		: SINT := 1;
	E_System_BHKW_Zustand_Status_Nachl_Stellventil	: SINT := 2;
	E_System_BHKW_Zustand_Status_Vorl_Stellventil	: SINT := 3;
	E_System_BHKW_Zustand_Status_Nachl_Pumpe		: SINT := 4;
	E_System_BHKW_Zustand_Status_Vorl_Pumpe			: SINT := 5;
	E_System_BHKW_Zustand_Status_Nachl_BHKW			: SINT := 6;
	E_System_BHKW_Zustand_Status_Vorl_BHKW			: SINT := 7;
	E_System_BHKW_Zustand_Status_Betrieb			: SINT := 8;
	E_System_BHKW_Zustand_Status_Betrieb_Sperre		: SINT := 9;
	E_System_BHKW_Zustand_Status_Ueberhitzt			: SINT := 10;
	E_System_BHKW_Zustand_Status_Stoerung			: SINT := 99;
END_VAR

// ---- Global Variables/Anlagen Variablen/Con_BSp.TcGVL
{attribute 'Tc2GvlVarNames'}
VAR_GLOBAL CONSTANT
	(* BSp_Zustand_Regelung_Modus *)
	E_BSp_Regelung_Modus_konst						: SINT := 0;
	E_BSp_Regelung_Modus_Laden_T_int				: SINT := 1;
	E_BSp_Regelung_Modus_Laden_T_ext				: SINT := 2;
	E_BSp_Regelung_Modus_Laden_dT					: SINT := 3;
	E_BSp_Regelung_Modus_Entladen_dT				: SINT := -3;
	E_BSp_Regelung_Modus_Entladen_T_int				: SINT := -1;
	E_BSp_Regelung_Modus_Entladen_T_ext				: SINT := -2;


	(* System_BSp_Zustand_Status *)
	E_System_BSp_Zustand_Status_Idle_Sperre			: SINT := 0;
	E_System_BSp_Zustand_Status_Betriebsbereit		: SINT := 1;
	E_System_BSp_Zustand_Status_Nachl_Stellventil	: SINT := 2;
	E_System_BSp_Zustand_Status_Vorl_Stellventil	: SINT := 3;
	E_System_BSp_Zustand_Status_Nachl_Pumpen		: SINT := 4;
	E_System_BSp_Zustand_Status_Vorl_Pumpen			: SINT := 5;
	E_System_BSp_Zustand_Status_Betrieb				: SINT := 8;
	E_System_BSp_Zustand_Status_Betrieb_Sperre		: SINT := 9;
	E_System_BSp_Zustand_Status_Stoerung			: SINT := 99;

	(* System_BSp_KueW_Zustand_Status *)
	E_System_BSp_KueW_Zustand_Status_Idle_Sperre	: SINT := 0;
	E_System_BSp_KueW_Zustand_Status_Betriebsbereit	: SINT := 1;
	E_System_BSp_KueW_Zustand_Status_Nachl			: SINT := 4;
	E_System_BSp_KueW_Zustand_Status_Vorl			: SINT := 5;
	E_System_BSp_KueW_Zustand_Status_Betrieb		: SINT := 8;
	E_System_BSp_KueW_Zustand_Status_Betrieb_Sperre	: SINT := 9;
	E_System_BSp_KueW_Zustand_Status_Stoerung		: SINT := 99;

	(* System_BSp_Verb_Zustand_Status *)
	E_System_BSp_Verb_Zustand_Status_Idle_Sperre	: SINT := 0;
	E_System_BSp_Verb_Zustand_Status_Betriebsbereit	: SINT := 1;
	E_System_BSp_Verb_Zustand_Status_Nachl_Pumpe	: SINT := 4;
	E_System_BSp_Verb_Zustand_Status_Vorl_Pumpe		: SINT := 5;
	E_System_BSp_Verb_Zustand_Status_Betrieb		: SINT := 8;
	E_System_BSp_Verb_Zustand_Status_Betrieb_Sperre	: SINT := 9;
	E_System_BSp_Verb_Zustand_Status_Stoerung		: SINT := 99;
END_VAR

// ---- Global Variables/Anlagen Variablen/Con_HO.TcGVL
{attribute 'Tc2GvlVarNames'}
VAR_GLOBAL CONSTANT
	(* HO_Zustand_Status *)
	E_HO_Zustand_Status_Idle_Sperre				: SINT := 0;
	E_HO_Zustand_Status_Betriebsbereit			: SINT := 1;
	E_HO_Zustand_Status_Nachl					: SINT := 2;
	E_HO_Zustand_Status_Vorl					: SINT := 3;
	E_HO_Zustand_Status_Betrieb					: SINT := 4;
	E_HO_Zustand_Status_Betrieb_Sperre			: SINT := 5;
	E_HO_Zustand_Status_Stoerung				: SINT := 99;

	(* System_HO_Zustand_Status *)
	E_System_HO_Zustand_Status_Idle_Sperre			: SINT := 0;
	E_System_HO_Zustand_Status_Betriebsbereit		: SINT := 1;
	E_System_HO_Zustand_Status_Nachl_Regelventil	: SINT := 2;
	E_System_HO_Zustand_Status_Vorl_Regelventil		: SINT := 3;
	E_System_HO_Zustand_Status_Nachl_Pumpe			: SINT := 4;
	E_System_HO_Zustand_Status_Vorl_Pumpe			: SINT := 5;
	(*E_System_HO_Zustand_Status_Nachl_HO			: SINT := 6;
	E_System_HO_Zustand_Status_Vorl_HO				: SINT := 7;	*)
	E_System_HO_Zustand_Status_Betrieb				: SINT := 8;
	E_System_HO_Zustand_Status_Betrieb_Sperre		: SINT := 9;
	E_System_HO_Zustand_Status_Stoerung				: SINT := 99;
END_VAR

// ---- Global Variables/Anlagen Variablen/Con_KKKW.TcGVL
{attribute 'Tc2GvlVarNames'}
VAR_GLOBAL CONSTANT
	(* KKKW_Zustand_Status *)
	E_KKKW_Zustand_Status_Idle_Sperre				: SINT := 0;
	E_KKKW_Zustand_Status_Betriebsbereit			: SINT := 1;
	E_KKKW_Zustand_Status_Nachl						: SINT := 2;
	E_KKKW_Zustand_Status_Vorl						: SINT := 3;
	E_KKKW_Zustand_Status_Betrieb					: SINT := 4;
	E_KKKW_Zustand_Status_Betrieb_Sperre			: SINT := 5;
	E_KKKW_Zustand_Status_Stoerung					: SINT := 99;

	(* System_KKKW_Zustand_Status *)
	E_System_KKKW_Zustand_Status_Idle_Sperre		: SINT := 0;
	E_System_KKKW_Zustand_Status_Betriebsbereit		: SINT := 1;
	E_System_KKKW_Zustand_Status_Nachl_Stellventil	: SINT := 2;
	E_System_KKKW_Zustand_Status_Vorl_Stellventil	: SINT := 3;
	E_System_KKKW_Zustand_Status_Nachl_Pumpe		: SINT := 4;
	E_System_KKKW_Zustand_Status_Vorl_Pumpe			: SINT := 5;
	(*E_System_KKKW_Zustand_Status_Nachl_KKKW		: SINT := 6;
	E_System_KKKW_Zustand_Status_Vorl_KKKW			: SINT := 7;	*)
	E_System_KKKW_Zustand_Status_Betrieb			: SINT := 8;
	E_System_KKKW_Zustand_Status_Betrieb_Sperre		: SINT := 9;
	E_System_KKKW_Zustand_Status_Stoerung			: SINT := 99;
END_VAR

// ---- Global Variables/Anlagen Variablen/Con_MVWW.TcGVL
{attribute 'Tc2GvlVarNames'}
VAR_GLOBAL CONSTANT
	(* KKWW_Zustand_Status *)
	E_MVWW_Zustand_Status_Idle_Sperre				: SINT := 0;
	E_MVWW_Zustand_Status_Betriebsbereit			: SINT := 1;
	E_MVWW_Zustand_Status_Nachl					: SINT := 2;
	E_MVWW_Zustand_Status_Vorl						: SINT := 3;
	E_MVWW_Zustand_Status_Betrieb					: SINT := 4;
	E_MVWW_Zustand_Status_Betrieb_Sperre			: SINT := 5;
	E_MVWW_Zustand_Status_Stoerung				: SINT := 99;

	(* System_KKWW_Zustand_Status *)
	E_System_MVWW_Zustand_Status_Idle_Sperre		: SINT := 0;
	E_System_MVWW_Zustand_Status_Betriebsbereit		: SINT := 1;
	E_System_MVWW_Zustand_Status_Nachl_Stellventil	: SINT := 2;
	E_System_MVWW_Zustand_Status_Vorl_Stellventil	: SINT := 3;
	E_System_MVWW_Zustand_Status_Nachl_Pumpe		: SINT := 4;
	E_System_MVWW_Zustand_Status_Vorl_Pumpe		: SINT := 5;
	(*E_System_MVWW_Zustand_Status_Nachl_KKWW		: SINT := 6;
	E_System_MVWW_Zustand_Status_Vorl_KKWW			: SINT := 7;	*)
	E_System_MVWW_Zustand_Status_Betrieb			: SINT := 8;
	E_System_MVWW_Zustand_Status_Betrieb_Sperre	: SINT := 9;
	E_System_MVWW_Zustand_Status_Stoerung			: SINT := 99;
END_VAR

// ---- Global Variables/Anlagen Variablen/Con_PU.TcGVL
{attribute 'Tc2GvlVarNames'}
VAR_GLOBAL CONSTANT
	(* Pumpe_Zustand_Status *)
	E_PU_Zustand_Status_Idle_Sperre			: SINT := 0;
	E_PU_Zustand_Status_Betriebsbereit		: SINT := 1;
	E_PU_Zustand_Status_Nachl				: SINT := 2;
	E_PU_Zustand_Status_Vorl				: SINT := 3;
	E_PU_Zustand_Status_Betrieb				: SINT := 4;
	E_PU_Zustand_Status_Betrieb_Sperre		: SINT := 5;
	E_PU_Zustand_Status_Stoerung			: SINT := 99;

	(* Pumpe_Zustand_Regelung_Modus *)
	E_PU_Regelung_Modus_P					: SINT := 0;
	E_PU_Regelung_Modus_dT					: SINT := 1;
	E_PU_Regelung_Modus_dT_invert			: SINT := 2;
	E_PU_Regelung_Modus_T_int				: SINT := 3;
	E_PU_Regelung_Modus_T_ext				: SINT := 4;
	E_PU_Regelung_Modus_dp_auto				: SINT := 5;
END_VAR

// ---- Global Variables/Anlagen Variablen/Con_SHZ.TcGVL
{attribute 'Tc2GvlVarNames'}
VAR_GLOBAL CONSTANT
	(* System_SHZ_Zustand_Status *)
	E_System_SHZ_Zustand_Status_Idle_Sperre					: SINT := 0;
	E_System_SHZ_Zustand_Status_Betriebsbereit				: SINT := 1;
	E_System_SHZ_Zustand_Status_Nachl_Pumpe					: SINT := 2;
	E_System_SHZ_Zustand_Status_Vorl_Pumpe					: SINT := 3;
	E_System_SHZ_Zustand_Status_Nachl_Regelventil			: SINT := 4;
	E_System_SHZ_Zustand_Status_Vorl_Regelventil			: SINT := 5;
	E_System_SHZ_Zustand_Status_Betrieb						: SINT := 6;
	E_System_SHZ_Zustand_Status_Betrieb_Sperre				: SINT := 7;
	E_System_SHZ_Zustand_Status_Stoerung					: SINT := 99;

	(* System_SHZ_Zustand_Regelung_Modus *)
	E_System_SHZ_Regelung_Modus_Automatik					: SINT := 0;
	E_System_SHZ_Regelung_Modus_Heizen_konst				: SINT := 1;
	E_System_SHZ_Regelung_Modus_Heizen_Kurve				: SINT := 2;
	E_System_SHZ_Regelung_Modus_Heizen_Kurve_Nachtabs		: SINT := 3;
	E_System_SHZ_Regelung_Modus_Kuehlen_konst				: SINT := -1;
	E_System_SHZ_Regelung_Modus_Kuehlen_Kurve				: SINT := -2;

END_VAR

// ---- Global Variables/Anlagen Variablen/Con_SV.TcGVL
{attribute 'Tc2GvlVarNames'}
VAR_GLOBAL CONSTANT
	(* Stellventil_Zustand_Status *)
	E_Stellventil_Zustand_Status_Stellungrueckmeldung0_Sperre	: SINT := 0;
	E_Stellventil_Zustand_Status_Stellungrueckmeldung0			: SINT := 1;
	E_Stellventil_Zustand_Stellungwechsel10						: SINT := 2;
	E_Stellventil_Zustand_Stellungwechsel01						: SINT := 3;
	E_Stellventil_Zustand_Status_Stellungrueckmeldung1			: SINT := 4;
	E_Stellventil_Zustand_Status_Stellungrueckmeldung1_Sperre	: SINT := 5;
	E_Stellventil_Zustand_Status_Stoerung						: SINT := 99;
END_VAR

// ---- Global Variables/Anlagen Variablen/Con_ThNTZ.TcGVL
{attribute 'Tc2GvlVarNames'}
VAR_GLOBAL CONSTANT
	(* ThNTZ_Zustand_Status *)
	E_ThNTZ_Zustand_Status_Idle_Sperre		: SINT := 0;
	E_ThNTZ_Zustand_Status_Betriebsbereit	: SINT := 1;
	E_ThNTZ_Zustand_Status_Betrieb			: SINT := 8;
	E_ThNTZ_Zustand_Status_Betrieb_Sperre	: SINT := 9;
	E_ThNTZ_Zustand_Status_Stoerung			: SINT := 99;

	(* ThNTZ_Zustand_Regelung_Modus *)
	E_ThNTZ_Regelung_Modus_Auto				: SINT := 0;
	E_ThNTZ_Regelung_Modus_T_Unten			: SINT := 1;
	E_ThNTZ_Regelung_Modus_T_Oben			: SINT := 2;
END_VAR

// ---- Global Variables/Anlagen Variablen/Con_WDT.TcGVL
{attribute 'Tc2GvlVarNames'}
VAR_GLOBAL CONSTANT
	(* System_WDT_Zustand_Status *)
	E_System_WDT_Zustand_Status_Idle_Sperre				: SINT := 0;
	E_System_WDT_Zustand_Status_Betriebsbereit			: SINT := 1;
	E_System_WDT_Zustand_Status_Nachl_Stellventil		: SINT := 2;
	E_System_WDT_Zustand_Status_Vorl_Stellventil		: SINT := 3;
	E_System_WDT_Zustand_Status_Nachl_Pumpe				: SINT := 4;
	E_System_WDT_Zustand_Status_Vorl_Pumpe				: SINT := 5;
	E_System_WDT_Zustand_Status_Nachl_Regelventil		: SINT := 6;
	E_System_WDT_Zustand_Status_Vorl_Regelventil		: SINT := 7;
	E_System_WDT_Zustand_Status_Betrieb					: SINT := 8;
	E_System_WDT_Zustand_Status_Betrieb_Sperre			: SINT := 9;
	E_System_WDT_Zustand_Status_Stoerung				: SINT := 99;

	(* System_WDT_Zustand_Regelung_Modus *)
	E_System_WDT_Regelung_Modus_Automatik						: SINT := 0;
	E_System_WDT_Regelung_Modus_Heizen_viaNetz_konst			: SINT := 1;
	E_System_WDT_Regelung_Modus_Heizen_viaNetz_Kurve			: SINT := 2;
	E_System_WDT_Regelung_Modus_Heizen_viaRueckkuehler_konst	: SINT := 3;
	E_System_WDT_Regelung_Modus_Heizen_viaRueckkuehler_Kurve	: SINT := 4;
	E_System_WDT_Regelung_Modus_Kuehlen_viaNetz_konst			: SINT := -1;
	E_System_WDT_Regelung_Modus_Kuehlen_viaNetz_Kurve			: SINT := -2;
	E_System_WDT_Regelung_Modus_Kuehlen_viaRueckkuehler_konst	: SINT := -3;
	E_System_WDT_Regelung_Modus_Kuehlen_viaRueckkuehler_Kurve	: SINT := -4;
END_VAR

// ---- Global Variables/Bus_Systeme/M_Bus.TcGVL
{attribute 'Tc2GvlVarNames'}
VAR_GLOBAL
	IN_Stromzaehler AT %I* 	: ST_KL6781inData22B;
	OUT_Stromzaehler AT %Q* : ST_KL6781outData22B;
	IN_WZaehler AT %I* 	: ST_KL6781inData22B;
	OUT_WZaehler AT %Q* : ST_KL6781outData22B;
	(*
			[1] ETA_3111U1006XHE321XXXXXXZ01, ELT_Zaehler_BHKW_321_01
			Primaer-Adresse = 1
			Seriennummer = 3999427
			[2] ETA_3111U1006XHE322XXXXXXZ01, ELT_Zaehler_BHKW_322_01
			Primaer-Adresse = 2
			Seriennummer = 3999432
			[3] ETA_3111U1006BEST001XXXXXXZ01, ELT_Zaehler_Buerotrakt_01
			Primaer-Adresse = 3
			Seriennummer = 120267
			[4] ETA_3111U1006BEST002XXXXXXZ01, ELT_Zaehler_Gebaede_01
			Primaer-Adresse = 4
			Seriennummer = 205684
			[5] ETA_3111U1006BEST003XXXXXXZ01, ELT_Zaehler_Halle_TGA_01
			Primaer-Adresse = 5
			Seriennummer = 120264
			[6] ETA_3111EG005BEST004XXXXXXZ01, ELT_Zaehler_Halle_Licht_01
			Primaer-Adresse = 6
			Seriennummer = 214516
			[7] ETA_3111U1006BEST007XXXXXXZ01, GAS_Zaehler BHKW_007_01
			Primaer-Adresse = 7
			Seriennummer = 42078747
			[8] ETA_3111U1006BEST008XXXXXXZ01, GAS_Zaehler BHKW_008_01
			Primaer-Adresse = 8
			Seriennummer = 42078748
			[9] ETA_3111U1006BEST071XXXXXXZ01, WAERME_Zaehler WP_945_4371_01
			Primaer-Adresse = 71
			Seriennummer = 67694371
			[10] ETA_3111U1006BEST072XXXXXXZ01, WAERME_Zaehler WP_945_4372_01
			Primaer-Adresse = 72
			Seriennummer = 67694372
	*)
	Kommunikation_MBus	: ST_MBUS_Communication;
	Komm_MBus_WZaehler	: ST_MBUS_Communication;

	Telegramm_WZ_Brennwerttherme			: ARRAY[1..cMBUS_MaxTelegrams] OF ST_MBus_Data2;
	Telegramm_WZ_BHKW_1						: ARRAY[1..cMBUS_MaxTelegrams] OF ST_MBus_Data2;
	Telegramm_WZ_BHKW_2						: ARRAY[1..cMBUS_MaxTelegrams] OF ST_MBus_Data2;
	Telegramm_WZ_Druckluftkompressor		: ARRAY[1..cMBUS_MaxTelegrams] OF ST_MBus_Data2;
	Telegramm_WZ_PWT_1						: ARRAY[1..cMBUS_MaxTelegrams] OF ST_MBus_Data2;
	Telegramm_WZ_Ofenkuehlung				: ARRAY[1..cMBUS_MaxTelegrams] OF ST_MBus_Data2;
	Telegramm_WZ_Abwaerme_Ofen_Abgasfackel	: ARRAY[1..cMBUS_MaxTelegrams] OF ST_MBus_Data2;

	Telegramm_SZ_BHKW_321		: ARRAY[1..cMBUS_MaxTelegrams] OF ST_MBus_Data2;
	Telegramm_SZ_BHKW_322		: ARRAY[1..cMBUS_MaxTelegrams] OF ST_MBus_Data2;
	Telegramm_SZ_Buerotrakt		: ARRAY[1..cMBUS_MaxTelegrams] OF ST_MBus_Data2;
	Telegramm_SZ_Gebaeude		: ARRAY[1..cMBUS_MaxTelegrams] OF ST_MBus_Data2;
	Telegramm_SZ_Halle_TGA		: ARRAY[1..cMBUS_MaxTelegrams] OF ST_MBus_Data2;
	Telegramm_SZ_Halle_Licht	: ARRAY[1..cMBUS_MaxTelegrams] OF ST_MBus_Data2;

	Telegramm_GZ_BHKW_321		: ARRAY[1..cMBUS_MaxTelegrams] OF ST_MBus_Data2;
	Telegramm_GZ_BHKW_322		: ARRAY[1..cMBUS_MaxTelegrams] OF ST_MBus_Data2;

	Telegramm_WZ_4371_WP_946	: ARRAY[1..cMBUS_MaxTelegrams] OF ST_MBus_Data2;
	Telegramm_WZ_4372_WP_946	: ARRAY[1..cMBUS_MaxTelegrams] OF ST_MBus_Data2;

END_VAR

// ---- Global Variables/Bus_Systeme/Profibus.TcGVL
{attribute 'Tc2GvlVarNames'}
VAR_GLOBAL
(*Master*)
(*Gerät 4 (CX5130-0121-M310), BOX 01*)
(*DP/DP-Kopppler*)
(*DP_State*)
(*
	R1_B01_PB_Zustand						AT %I*: USINT;
(*Daten*)
	R1_B01_StatusModule_I_Byte_1			AT %I*: USINT;
	R1_B01_StatusModule_I_Byte_2			AT %I*: USINT;
	R1_B01_StatusModule_I_Byte_5			AT %I*: USINT;
	R1_B01_StatusModule_I_Byte_6			AT %I*: USINT;
	R1_B01_ControlModule_O					AT %Q* :ARRAY [0..4] OF USINT;
	R1_B01_VolumeFlow_I						AT %I* :UDINT;
	R1_B01_PumpLiquidTemp_I					AT %I* :UDINT;
	R1_B01_OperationTime_I					AT %I* :UDINT;
	R1_B01_ActualSetpoint_I					AT %I* :UDINT;
	R1_B01_Frequency_I						AT %I* :UDINT;
	R1_B01_UserSetpoint_I					AT %I* :UDINT;
	R1_B01_DiffPressure_I					AT %I* :UDINT;
	R1_B01_RemoteTemp2						AT %I* :UDINT;
	R1_B01_HeatEnergyCounter_I				AT %I* :UDINT;
	R1_B01_HeatDiffTemp						AT %I* :UDINT;
	R1_B01_HeatPower						AT %I* :UDINT;  (* B0_SequenceNumber(1),B1AddressGenib(30),B2Class(11),B3Operation_Lenght(1),B4Data1(ID.34),Data(B5-B8) *)
	R1_B01_DirectDataReques_Temp_Geni		AT %Q* :PB_GenibusType;		(*ARRAY [0..8] OF USINT := 1, 255, 11, 1, 34, 0, 0, 0, 0;*)
	R1_B01_DirectDataReply_Temp_Geni		AT %I* :PB_GenibusType;		(*ARRAY [0..8] OF USINT;*)



	R1_B01_NumberOfStarts					AT %I*	: 	UDINT;
	R1_B01_ActualSetpoint					AT %I*	:	UDINT;
	R1_B01_OperationTime					AT %I*	: 	UDINT;
	R1_B01_Speed							AT %I*	:	UDINT;
	R1_B01_Energy							AT %I*	: 	UDINT;
	R1_B01_Power							AT %I*	:	UDINT;
	R1_B01_PowerElectronicsTemp				AT %I*	:	UDINT;
	R1_B01_FaultCode						AT %I*	:	USINT;
	R1_B01_Volume							AT %I*	:	UDINT;
	R1_B01_WarningCode						AT %I*	:	USINT;

(*Gerät 4 (CX5130-0121-M310), BOX 02*)
(*DP/DP-Kopppler*)
(*DP_State*)
	R1_B02_PB_Zustand						AT %I*: USINT;
(*Daten*)
	R1_B02_StatusModule_I_Byte_1			AT %I*: USINT;
	R1_B02_StatusModule_I_Byte_2			AT %I*: USINT;
	R1_B02_StatusModule_I_Byte_5			AT %I*: USINT;
	R1_B02_StatusModule_I_Byte_6			AT %I*: USINT;
	R1_B02_ControlModule_O					AT %Q* :ARRAY [0..4] OF USINT;
	R1_B02_VolumeFlow_I						AT %I* :UDINT;
	R1_B02_PumpLiquidTemp_I					AT %I* :UDINT;
	R1_B02_OperationTime_I					AT %I* :UDINT;
	R1_B02_ActualSetpoint_I					AT %I* :UDINT;
	R1_B02_Frequency_I						AT %I* :UDINT;
	R1_B02_UserSetpoint_I					AT %I* :UDINT;
	R1_B02_DiffPressure_I					AT %I* :UDINT;
	R1_B02_RemoteTemp2						AT %I* :UDINT;
	R1_B02_HeatEnergyCounter_I				AT %I* :UDINT;
	R1_B02_HeatDiffTemp						AT %I* :UDINT;
	R1_B02_HeatPower						AT %I* :UDINT;(* B0_SequenceNumber(1),B1AddressGenib(30),B2Class(11),B3Operation_Lenght(1),B4Data1(ID.34),Data(B5-B8) *)
	R1_B02_DirectDataReques_Temp_Geni		AT %Q* :PB_GenibusType;
	R1_B02_DirectDataReply_Temp_Geni		AT %I* :PB_GenibusType;


	R1_B02_NumberOfStarts					AT %I*	: 	UDINT;
	R1_B02_ActualSetpoint					AT %I*	:	UDINT;
	R1_B02_OperationTime					AT %I*	: 	UDINT;
	R1_B02_Speed							AT %I*	:	UDINT;
	R1_B02_Energy							AT %I*	: 	UDINT;
	R1_B02_Power							AT %I*	:	UDINT;
	R1_B02_PowerElectronicsTemp				AT %I*	:	UDINT;
	R1_B02_FaultCode						AT %I*	:	USINT;
	R1_B02_Volume							AT %I*	:	UDINT;
	R1_B02_WarningCode						AT %I*	:	USINT;

(*Gerät 4 (CX5130-0121-M310), BOX 03*)
(*DP/DP-Kopppler*)
(*DP_State*)
	R1_B03_PB_Zustand						AT %I*: USINT;
(*Daten*)
	R1_B03_StatusModule_I_Byte_1			AT %I*: USINT;
	R1_B03_StatusModule_I_Byte_2			AT %I*: USINT;
	R1_B03_StatusModule_I_Byte_5			AT %I*: USINT;
	R1_B03_StatusModule_I_Byte_6			AT %I*: USINT;
	R1_B03_ControlModule_O					AT %Q* :ARRAY [0..4] OF USINT;
	R1_B03_VolumeFlow_I						AT %I* :UDINT;
	R1_B03_PumpLiquidTemp_I					AT %I* :UDINT;
	R1_B03_OperationTime_I					AT %I* :UDINT;
	R1_B03_ActualSetpoint_I					AT %I* :UDINT;
	R1_B03_Frequency_I						AT %I* :UDINT;
	R1_B03_UserSetpoint_I					AT %I* :UDINT;
	R1_B03_DiffPressure_I					AT %I* :UDINT;
	R1_B03_RemoteTemp2						AT %I* :UDINT;
	R1_B03_HeatEnergyCounter_I				AT %I* :UDINT;
	R1_B03_HeatDiffTemp						AT %I* :UDINT;
	R1_B03_HeatPower						AT %I* :UDINT;(* B0_SequenceNumber(1),B1AddressGenib(30),B2Class(11),B3Operation_Lenght(1),B4Data1(ID.34),Data(B5-B8) *)
	R1_B03_DirectDataReques_Temp_Geni		AT %Q* :PB_GenibusType;
	R1_B03_DirectDataReply_Temp_Geni		AT %I* :PB_GenibusType;

	R1_B03_NumberOfStarts					AT %I*	: 	UDINT;
	R1_B03_ActualSetpoint					AT %I*	:	UDINT;
	R1_B03_OperationTime					AT %I*	: 	UDINT;
	R1_B03_Speed							AT %I*	:	UDINT;
	R1_B03_Energy							AT %I*	: 	UDINT;
	R1_B03_Power							AT %I*	:	UDINT;
	R1_B03_PowerElectronicsTemp				AT %I*	:	UDINT;
	R1_B03_FaultCode						AT %I*	:	USINT;
	R1_B03_Volume							AT %I*	:	UDINT;
	R1_B03_WarningCode						AT %I*	:	USINT;

(*Gerät 4 (CX5130-0121-M310), BOX 04*)
(*DP/DP-Kopppler*)
(*DP_State*)
	R1_B04_PB_Zustand						AT %I*: USINT;
(*Daten*)
	R1_B04_StatusModule_I_Byte_1			AT %I*: USINT;
	R1_B04_StatusModule_I_Byte_2			AT %I*: USINT;
	R1_B04_StatusModule_I_Byte_5			AT %I*: USINT;
	R1_B04_StatusModule_I_Byte_6			AT %I*: USINT;
	R1_B04_ControlModule_O					AT %Q* :ARRAY [0..4] OF USINT;
	R1_B04_VolumeFlow_I						AT %I* :UDINT;
	R1_B04_PumpLiquidTemp_I					AT %I* :UDINT;
	R1_B04_OperationTime_I					AT %I* :UDINT;
	R1_B04_ActualSetpoint_I					AT %I* :UDINT;
	R1_B04_Frequency_I						AT %I* :UDINT;
	R1_B04_UserSetpoint_I					AT %I* :UDINT;
	R1_B04_DiffPressure_I					AT %I* :UDINT;
	R1_B04_RemoteTemp2						AT %I* :UDINT;
	R1_B04_HeatEnergyCounter_I				AT %I* :UDINT;
	R1_B04_HeatDiffTemp						AT %I* :UDINT;
	R1_B04_HeatPower						AT %I* :UDINT;(* B0_SequenceNumber(1),B1AddressGenib(30),B2Class(11),B3Operation_Lenght(1),B4Data1(ID.34),Data(B5-B8) *)
	R1_B04_DirectDataReques_Temp_Geni		AT %Q* :PB_GenibusType;
	R1_B04_DirectDataReply_Temp_Geni		AT %I* :PB_GenibusType;


	R1_B04_NumberOfStarts					AT %I*	: 	UDINT;
	R1_B04_ActualSetpoint					AT %I*	:	UDINT;
	R1_B04_OperationTime					AT %I*	: 	UDINT;
	R1_B04_Speed							AT %I*	:	UDINT;
	R1_B04_Energy							AT %I*	: 	UDINT;
	R1_B04_Power							AT %I*	:	UDINT;
	R1_B04_PowerElectronicsTemp				AT %I*	:	UDINT;
	R1_B04_FaultCode						AT %I*	:	USINT;
	R1_B04_Volume							AT %I*	:	UDINT;
	R1_B04_WarningCode						AT %I*	:	USINT;


(*Gerät 4 (CX5130-0121-M310), BOX 05*)
(*DP/DP-Kopppler*)
(*DP_State*)
	R1_B05_PB_Zustand						AT %I*: USINT;
(*Daten*)
	R1_B05_StatusModule_I_Byte_1			AT %I*: USINT;
	R1_B05_StatusModule_I_Byte_2			AT %I*: USINT;
	R1_B05_StatusModule_I_Byte_5			AT %I*: USINT;
	R1_B05_StatusModule_I_Byte_6			AT %I*: USINT;
	R1_B05_ControlModule_O					AT %Q* :ARRAY [0..4] OF USINT;
	R1_B05_VolumeFlow_I						AT %I* :UDINT;
	R1_B05_PumpLiquidTemp_I					AT %I* :UDINT;
	R1_B05_OperationTime_I					AT %I* :UDINT;
	R1_B05_ActualSetpoint_I					AT %I* :UDINT;
	R1_B05_Frequency_I						AT %I* :UDINT;
	R1_B05_UserSetpoint_I					AT %I* :UDINT;
	R1_B05_DiffPressure_I					AT %I* :UDINT;
	R1_B05_RemoteTemp2						AT %I* :UDINT;
	R1_B05_HeatEnergyCounter_I				AT %I* :UDINT;
	R1_B05_HeatDiffTemp						AT %I* :UDINT;
	R1_B05_HeatPower						AT %I* :UDINT;(* B0_SequenceNumber(1),B1AddressGenib(30),B2Class(11),B3Operation_Lenght(1),B4Data1(ID.34),Data(B5-B8) *)
	R1_B05_DirectDataReques_Temp_Geni		AT %Q* :PB_GenibusType;
	R1_B05_DirectDataReply_Temp_Geni		AT %I* :PB_GenibusType;

	R1_B05_NumberOfStarts					AT %I*	: 	UDINT;
	R1_B05_ActualSetpoint					AT %I*	:	UDINT;
	R1_B05_OperationTime					AT %I*	: 	UDINT;
	R1_B05_Speed							AT %I*	:	UDINT;
	R1_B05_Energy							AT %I*	: 	UDINT;
	R1_B05_Power							AT %I*	:	UDINT;
	R1_B05_PowerElectronicsTemp				AT %I*	:	UDINT;
	R1_B05_FaultCode						AT %I*	:	USINT;
	R1_B05_Volume							AT %I*	:	UDINT;
	R1_B05_WarningCode						AT %I*	:	USINT;


(*Gerät 4 (CX5130-0121-M310), BOX 06*)
(*DP/DP-Kopppler*)
(*DP_State*)
	R1_B06_PB_Zustand						AT %I*: USINT;
(*Daten*)
	R1_B06_StatusModule_I_Byte_1			AT %I*: USINT;
	R1_B06_StatusModule_I_Byte_2			AT %I*: USINT;
	R1_B06_StatusModule_I_Byte_5			AT %I*: USINT;
	R1_B06_StatusModule_I_Byte_6			AT %I*: USINT;
	R1_B06_ControlModule_O					AT %Q* :ARRAY [0..4] OF USINT;
	R1_B06_VolumeFlow_I						AT %I* :UDINT;
	R1_B06_PumpLiquidTemp_I					AT %I* :UDINT;
	R1_B06_OperationTime_I					AT %I* :UDINT;
	R1_B06_ActualSetpoint_I					AT %I* :UDINT;
	R1_B06_Frequency_I						AT %I* :UDINT;
	R1_B06_UserSetpoint_I					AT %I* :UDINT;
	R1_B06_DiffPressure_I					AT %I* :UDINT;
	R1_B06_RemoteTemp2						AT %I* :UDINT;
	R1_B06_HeatEnergyCounter_I				AT %I* :UDINT;
	R1_B06_HeatDiffTemp						AT %I* :UDINT;
	R1_B06_HeatPower						AT %I* :UDINT;(* B0_SequenceNumber(1),B1AddressGenib(30),B2Class(11),B3Operation_Lenght(1),B4Data1(ID.34),Data(B5-B8) *)
	R1_B06_DirectDataReques_Temp_Geni		AT %Q* :PB_GenibusType;
	R1_B06_DirectDataReply_Temp_Geni		AT %I* :PB_GenibusType;

	R1_B06_NumberOfStarts					AT %I*	: 	UDINT;
	R1_B06_ActualSetpoint					AT %I*	:	UDINT;
	R1_B06_OperationTime					AT %I*	: 	UDINT;
	R1_B06_Speed							AT %I*	:	UDINT;
	R1_B06_Energy							AT %I*	: 	UDINT;
	R1_B06_Power							AT %I*	:	UDINT;
	R1_B06_PowerElectronicsTemp				AT %I*	:	UDINT;
	R1_B06_FaultCode						AT %I*	:	USINT;
	R1_B06_Volume							AT %I*	:	UDINT;
	R1_B06_WarningCode						AT %I*	:	USINT;

(*Gerät 4 (CX5130-0121-M310), BOX 07*)                           (*Pumpe entfallen*)
(*DP/DP-Kopppler*)
(*DP_State*)
	R1_B07_PB_Zustand						AT %I*: USINT;
(*Daten*)
	R1_B07_StatusModule_I_Byte_1			AT %I*: USINT;
	R1_B07_StatusModule_I_Byte_2			AT %I*: USINT;
	R1_B07_StatusModule_I_Byte_5			AT %I*: USINT;
	R1_B07_StatusModule_I_Byte_6			AT %I*: USINT;
	R1_B07_ControlModule_O					AT %Q* :ARRAY [0..4] OF USINT;
	R1_B07_VolumeFlow_I						AT %I* :UDINT;
	R1_B07_PumpLiquidTemp_I					AT %I* :UDINT;
	R1_B07_OperationTime_I					AT %I* :UDINT;
	R1_B07_ActualSetpoint_I					AT %I* :UDINT;
	R1_B07_Frequency_I						AT %I* :UDINT;
	R1_B07_UserSetpoint_I					AT %I* :UDINT;
	R1_B07_DiffPressure_I					AT %I* :UDINT;
	R1_B07_RemoteTemp2						AT %I* :UDINT;
	R1_B07_HeatEnergyCounter_I				AT %I* :UDINT;
	R1_B07_HeatDiffTemp						AT %I* :UDINT;
	R1_B07_HeatPower						AT %I* :UDINT;

	R1_B07_NumberOfStarts					AT %I*	: 	UDINT;
	R1_B07_ActualSetpoint					AT %I*	:	UDINT;
	R1_B07_OperationTime					AT %I*	: 	UDINT;
	R1_B07_Speed							AT %I*	:	UDINT;
	R1_B07_Energy							AT %I*	: 	UDINT;
	R1_B07_Power							AT %I*	:	UDINT;
	R1_B07_PowerElectronicsTemp				AT %I*	:	UDINT;
	R1_B07_FaultCode						AT %I*	:	USINT;
	R1_B07_Volume							AT %I*	:	UDINT;
	R1_B07_WarningCode						AT %I*	:	USINT;


(*Gerät 4 (CX5130-0121-M310), BOX 08*)							  (*Pumpe entfallen*)
(*DP/DP-Kopppler*)
(*DP_State*)
	R1_B08_PB_Zustand						AT %I*: USINT;
(*Daten*)
	R1_B08_StatusModule_I_Byte_1			AT %I*: USINT;
	R1_B08_StatusModule_I_Byte_2			AT %I*: USINT;
	R1_B08_StatusModule_I_Byte_5			AT %I*: USINT;
	R1_B08_StatusModule_I_Byte_6			AT %I*: USINT;
	R1_B08_ControlModule_O					AT %Q* :ARRAY [0..4] OF USINT;
	R1_B08_VolumeFlow_I						AT %I* :UDINT;
	R1_B08_PumpLiquidTemp_I					AT %I* :UDINT;
	R1_B08_OperationTime_I					AT %I* :UDINT;
	R1_B08_ActualSetpoint_I					AT %I* :UDINT;
	R1_B08_Frequency_I						AT %I* :UDINT;
	R1_B08_UserSetpoint_I					AT %I* :UDINT;
	R1_B08_DiffPressure_I					AT %I* :UDINT;
	R1_B08_RemoteTemp2						AT %I* :UDINT;
	R1_B08_HeatEnergyCounter_I				AT %I* :UDINT;
	R1_B08_HeatDiffTemp						AT %I* :UDINT;
	R1_B08_HeatPower						AT %I* :UDINT;

	R1_B08_NumberOfStarts					AT %I*	: 	UDINT;
	R1_B08_ActualSetpoint					AT %I*	:	UDINT;
	R1_B08_OperationTime					AT %I*	: 	UDINT;
	R1_B08_Speed							AT %I*	:	UDINT;
	R1_B08_Energy							AT %I*	: 	UDINT;
	R1_B08_Power							AT %I*	:	UDINT;
	R1_B08_PowerElectronicsTemp				AT %I*	:	UDINT;
	R1_B08_FaultCode						AT %I*	:	USINT;
	R1_B08_Volume							AT %I*	:	UDINT;
	R1_B08_WarningCode						AT %I*	:	USINT;

(*Gerät 4 (CX5130-0121-M310), BOX 09*)
(*DP/DP-Kopppler*)
(*DP_State*)
	R1_B09_PB_Zustand						AT %I*: USINT;
(*Daten*)
	R1_B09_StatusModule_I_Byte_1			AT %I*: USINT;
	R1_B09_StatusModule_I_Byte_2			AT %I*: USINT;
	R1_B09_StatusModule_I_Byte_5			AT %I*: USINT;
	R1_B09_StatusModule_I_Byte_6			AT %I*: USINT;
	R1_B09_ControlModule_O					AT %Q* :ARRAY [0..4] OF USINT;
	R1_B09_VolumeFlow_I						AT %I* :UDINT;
	R1_B09_PumpLiquidTemp_I					AT %I* :UDINT;
	R1_B09_OperationTime_I					AT %I* :UDINT;
	R1_B09_ActualSetpoint_I					AT %I* :UDINT;
	R1_B09_Frequency_I						AT %I* :UDINT;
	R1_B09_UserSetpoint_I					AT %I* :UDINT;
	R1_B09_DiffPressure_I					AT %I* :UDINT;
	R1_B09_RemoteTemp2						AT %I* :UDINT;
	R1_B09_HeatEnergyCounter_I				AT %I* :UDINT;
	R1_B09_HeatDiffTemp						AT %I* :UDINT;
	R1_B09_HeatPower						AT %I* :UDINT;(* B0_SequenceNumber(1),B1AddressGenib(30),B2Class(11),B3Operation_Lenght(1),B4Data1(ID.34),Data(B5-B8) *)
	R1_B09_DirectDataReques_Temp_Geni		AT %Q* :PB_GenibusType;
	R1_B09_DirectDataReply_Temp_Geni		AT %I* :PB_GenibusType;

	R1_B09_NumberOfStarts					AT %I*	: 	UDINT;
	R1_B09_ActualSetpoint					AT %I*	:	UDINT;
	R1_B09_OperationTime					AT %I*	: 	UDINT;
	R1_B09_Speed							AT %I*	:	UDINT;
	R1_B09_Energy							AT %I*	: 	UDINT;
	R1_B09_Power							AT %I*	:	UDINT;
	R1_B09_PowerElectronicsTemp				AT %I*	:	UDINT;
	R1_B09_FaultCode						AT %I*	:	USINT;
	R1_B09_Volume							AT %I*	:	UDINT;
	R1_B09_WarningCode						AT %I*	:	USINT;

(*Gerät 4 (CX5130-0121-M310), BOX 10*)
(*DP/DP-Kopppler*)
(*DP_State*)
	R1_B10_PB_Zustand						AT %I*: USINT;
(*Daten*)
	R1_B10_StatusModule_I_Byte_1			AT %I*: USINT;
	R1_B10_StatusModule_I_Byte_2			AT %I*: USINT;
	R1_B10_StatusModule_I_Byte_5			AT %I*: USINT;
	R1_B10_StatusModule_I_Byte_6			AT %I*: USINT;
	R1_B10_ControlModule_O					AT %Q* :ARRAY [0..4] OF USINT;
	R1_B10_VolumeFlow_I						AT %I* :UDINT;
	R1_B10_PumpLiquidTemp_I					AT %I* :UDINT;
	R1_B10_OperationTime_I					AT %I* :UDINT;
	R1_B10_ActualSetpoint_I					AT %I* :UDINT;
	R1_B10_Frequency_I						AT %I* :UDINT;
	R1_B10_UserSetpoint_I					AT %I* :UDINT;
	R1_B10_DiffPressure_I					AT %I* :UDINT;
	R1_B10_RemoteTemp2						AT %I* :UDINT;
	R1_B10_HeatEnergyCounter_I				AT %I* :UDINT;
	R1_B10_HeatDiffTemp						AT %I* :UDINT;
	R1_B10_HeatPower						AT %I* :UDINT;(* B0_SequenceNumber(1),B1AddressGenib(30),B2Class(11),B3Operation_Lenght(1),B4Data1(ID.34),Data(B5-B8) *)
	R1_B10_DirectDataReques_Temp_Geni		AT %Q* :PB_GenibusType;
	R1_B10_DirectDataReply_Temp_Geni		AT %I* :PB_GenibusType;

	R1_B10_NumberOfStarts					AT %I*	: 	UDINT;
	R1_B10_ActualSetpoint					AT %I*	:	UDINT;
	R1_B10_OperationTime					AT %I*	: 	UDINT;
	R1_B10_Speed							AT %I*	:	UDINT;
	R1_B10_Energy							AT %I*	: 	UDINT;
	R1_B10_Power							AT %I*	:	UDINT;
	R1_B10_PowerElectronicsTemp				AT %I*	:	UDINT;
	R1_B10_FaultCode						AT %I*	:	USINT;
	R1_B10_Volume							AT %I*	:	UDINT;
	R1_B10_WarningCode						AT %I*	:	USINT;

(*Gerät 4 (CX5130-0121-M310), BOX 11*)
(*DP/DP-Kopppler*)
(*DP_State*)
	R1_B11_PB_Zustand						AT %I*: USINT;
(*Daten*)
	R1_B11_StatusModule_I_Byte_1			AT %I*: USINT;
	R1_B11_StatusModule_I_Byte_2			AT %I*: USINT;
	R1_B11_StatusModule_I_Byte_5			AT %I*: USINT;
	R1_B11_StatusModule_I_Byte_6			AT %I*: USINT;
	R1_B11_ControlModule_O					AT %Q* :ARRAY [0..4] OF USINT;
	R1_B11_VolumeFlow_I						AT %I* :UDINT;
	R1_B11_PumpLiquidTemp_I					AT %I* :UDINT;
	R1_B11_OperationTime_I					AT %I* :UDINT;
	R1_B11_ActualSetpoint_I					AT %I* :UDINT;
	R1_B11_Frequency_I						AT %I* :UDINT;
	R1_B11_UserSetpoint_I					AT %I* :UDINT;
	R1_B11_DiffPressure_I					AT %I* :UDINT;
	R1_B11_RemoteTemp2						AT %I* :UDINT;
	R1_B11_HeatEnergyCounter_I				AT %I* :UDINT;
	R1_B11_HeatDiffTemp						AT %I* :UDINT;
	R1_B11_HeatPower						AT %I* :UDINT;(* B0_SequenceNumber(1),B1AddressGenib(30),B2Class(11),B3Operation_Lenght(1),B4Data1(ID.34),Data(B5-B8) *)
	R1_B11_DirectDataReques_Temp_Geni		AT %Q* :PB_GenibusType;
	R1_B11_DirectDataReply_Temp_Geni		AT %I* :PB_GenibusType;


	R1_B11_NumberOfStarts					AT %I*	: 	UDINT;
	R1_B11_ActualSetpoint					AT %I*	:	UDINT;
	R1_B11_OperationTime					AT %I*	: 	UDINT;
	R1_B11_Speed							AT %I*	:	UDINT;
	R1_B11_Energy							AT %I*	: 	UDINT;
	R1_B11_Power							AT %I*	:	UDINT;
	R1_B11_PowerElectronicsTemp				AT %I*	:	UDINT;
	R1_B11_FaultCode						AT %I*	:	USINT;
	R1_B11_Volume							AT %I*	:	UDINT;
	R1_B11_WarningCode						AT %I*	:	USINT;

(*Gerät 4 (CX5130-0121-M310), BOX 12*)								  (*Pumpe entfallen*)
(*DP/DP-Kopppler*)
(*DP_State*)
	R1_B12_PB_Zustand						AT %I*: USINT;
(*Daten*)
	R1_B12_StatusModule_I_Byte_1			AT %I*: USINT;
	R1_B12_StatusModule_I_Byte_2			AT %I*: USINT;
	R1_B12_StatusModule_I_Byte_5			AT %I*: USINT;
	R1_B12_StatusModule_I_Byte_6			AT %I*: USINT;
	R1_B12_ControlModule_O					AT %Q* :ARRAY [0..4] OF USINT;
	R1_B12_VolumeFlow_I						AT %I* :UDINT;
	R1_B12_PumpLiquidTemp_I					AT %I* :UDINT;
	R1_B12_OperationTime_I					AT %I* :UDINT;
	R1_B12_ActualSetpoint_I					AT %I* :UDINT;
	R1_B12_Frequency_I						AT %I* :UDINT;
	R1_B12_UserSetpoint_I					AT %I* :UDINT;
	R1_B12_DiffPressure_I					AT %I* :UDINT;
	R1_B12_RemoteTemp2						AT %I* :UDINT;
	R1_B12_HeatEnergyCounter_I				AT %I* :UDINT;
	R1_B12_HeatDiffTemp						AT %I* :UDINT;
	R1_B12_HeatPower						AT %I* :UDINT;

(*Gerät 4 (CX5130-0121-M310), BOX 13*)
(*DP/DP-Kopppler*)
(*DP_State*)
	R1_B13_PB_Zustand						AT %I*: USINT;
(*Daten*)
	R1_B13_StatusModule_I_Byte_1			AT %I*: USINT;
	R1_B13_StatusModule_I_Byte_2			AT %I*: USINT;
	R1_B13_StatusModule_I_Byte_5			AT %I*: USINT;
	R1_B13_StatusModule_I_Byte_6			AT %I*: USINT;
	R1_B13_ControlModule_O					AT %Q* :ARRAY [0..4] OF USINT;
	R1_B13_VolumeFlow_I						AT %I* :UDINT;
	R1_B13_PumpLiquidTemp_I					AT %I* :UDINT;
	R1_B13_OperationTime_I					AT %I* :UDINT;
	R1_B13_ActualSetpoint_I					AT %I* :UDINT;
	R1_B13_Frequency_I						AT %I* :UDINT;
	R1_B13_UserSetpoint_I					AT %I* :UDINT;
	R1_B13_DiffPressure_I					AT %I* :UDINT;
	R1_B13_RemoteTemp2						AT %I* :UDINT;
	R1_B13_HeatEnergyCounter_I				AT %I* :UDINT;
	R1_B13_HeatDiffTemp						AT %I* :UDINT;
	R1_B13_HeatPower						AT %I* :UDINT;(* B0_SequenceNumber(1),B1AddressGenib(30),B2Class(11),B3Operation_Lenght(1),B4Data1(ID.34),Data(B5-B8) *)
	R1_B13_DirectDataReques_Temp_Geni		AT %Q* :PB_GenibusType;
	R1_B13_DirectDataReply_Temp_Geni		AT %I* :PB_GenibusType;


	R1_B13_NumberOfStarts					AT %I*	: 	UDINT;
	R1_B13_ActualSetpoint					AT %I*	:	UDINT;
	R1_B13_OperationTime					AT %I*	: 	UDINT;
	R1_B13_Speed							AT %I*	:	UDINT;
	R1_B13_Energy							AT %I*	: 	UDINT;
	R1_B13_Power							AT %I*	:	UDINT;
	R1_B13_PowerElectronicsTemp				AT %I*	:	UDINT;
	R1_B13_FaultCode						AT %I*	:	USINT;
	R1_B13_Volume							AT %I*	:	UDINT;
	R1_B13_WarningCode						AT %I*	:	USINT;

(*Gerät 4 (CX5130-0121-M310), BOX 14*)
(*DP/DP-Kopppler*)
(*DP_State*)
	R1_B14_PB_Zustand						AT %I*: USINT;
(*Daten*)
	R1_B14_StatusModule_I_Byte_1			AT %I*: USINT;
	R1_B14_StatusModule_I_Byte_2			AT %I*: USINT;
	R1_B14_StatusModule_I_Byte_5			AT %I*: USINT;
	R1_B14_StatusModule_I_Byte_6			AT %I*: USINT;
	R1_B14_ControlModule_O					AT %Q* :ARRAY [0..4] OF USINT;
	R1_B14_VolumeFlow_I						AT %I* :UDINT;
	R1_B14_PumpLiquidTemp_I					AT %I* :UDINT;
	R1_B14_OperationTime_I					AT %I* :UDINT;
	R1_B14_ActualSetpoint_I					AT %I* :UDINT;
	R1_B14_Frequency_I						AT %I* :UDINT;
	R1_B14_UserSetpoint_I					AT %I* :UDINT;
	R1_B14_DiffPressure_I					AT %I* :UDINT;
	R1_B14_RemoteTemp2						AT %I* :UDINT;
	R1_B14_HeatEnergyCounter_I				AT %I* :UDINT;
	R1_B14_HeatDiffTemp						AT %I* :UDINT;
	R1_B14_HeatPower						AT %I* :UDINT;(* B0_SequenceNumber(1),B1AddressGenib(30),B2Class(11),B3Operation_Lenght(1),B4Data1(ID.34),Data(B5-B8) *)
	R1_B14_DirectDataReques_Temp_Geni		AT %Q* :PB_GenibusType;
	R1_B14_DirectDataReply_Temp_Geni		AT %I* :PB_GenibusType;


	R1_B14_NumberOfStarts					AT %I*	: 	UDINT;
	R1_B14_ActualSetpoint					AT %I*	:	UDINT;
	R1_B14_OperationTime					AT %I*	: 	UDINT;
	R1_B14_Speed							AT %I*	:	UDINT;
	R1_B14_Energy							AT %I*	: 	UDINT;
	R1_B14_Power							AT %I*	:	UDINT;
	R1_B14_PowerElectronicsTemp				AT %I*	:	UDINT;
	R1_B14_FaultCode						AT %I*	:	USINT;
	R1_B14_Volume							AT %I*	:	UDINT;
	R1_B14_WarningCode						AT %I*	:	USINT;

(*Gerät 4 (CX5130-0121-M310), BOX 15*)
(*DP/DP-Kopppler*)
(*DP_State*)
	R1_B15_PB_Zustand						AT %I*: USINT;
(*Daten*)
	R1_B15_StatusModule_I_Byte_1			AT %I*: USINT;
	R1_B15_StatusModule_I_Byte_2			AT %I*: USINT;
	R1_B15_StatusModule_I_Byte_5			AT %I*: USINT;
	R1_B15_StatusModule_I_Byte_6			AT %I*: USINT;
	R1_B15_ControlModule_O					AT %Q* :ARRAY [0..4] OF USINT;
	R1_B15_VolumeFlow_I						AT %I* :UDINT;
	R1_B15_PumpLiquidTemp_I					AT %I* :UDINT;
	R1_B15_OperationTime_I					AT %I* :UDINT;
	R1_B15_ActualSetpoint_I					AT %I* :UDINT;
	R1_B15_Frequency_I						AT %I* :UDINT;
	R1_B15_UserSetpoint_I					AT %I* :UDINT;
	R1_B15_DiffPressure_I					AT %I* :UDINT;
	R1_B15_RemoteTemp2						AT %I* :UDINT;
	R1_B15_HeatEnergyCounter_I				AT %I* :UDINT;
	R1_B15_HeatDiffTemp						AT %I* :UDINT;
	R1_B15_HeatPower						AT %I* :UDINT;(* B0_SequenceNumber(1),B1AddressGenib(30),B2Class(11),B3Operation_Lenght(1),B4Data1(ID.34),Data(B5-B8) *)
	R1_B15_DirectDataReques_Temp_Geni		AT %Q* :PB_GenibusType;
	R1_B15_DirectDataReply_Temp_Geni		AT %I* :PB_GenibusType;


	R1_B15_NumberOfStarts					AT %I*	: 	UDINT;
	R1_B15_ActualSetpoint					AT %I*	:	UDINT;
	R1_B15_OperationTime					AT %I*	: 	UDINT;
	R1_B15_Speed							AT %I*	:	UDINT;
	R1_B15_Energy							AT %I*	: 	UDINT;
	R1_B15_Power							AT %I*	:	UDINT;
	R1_B15_PowerElectronicsTemp				AT %I*	:	UDINT;
	R1_B15_FaultCode						AT %I*	:	USINT;
	R1_B15_Volume							AT %I*	:	UDINT;
	R1_B15_WarningCode						AT %I*	:	USINT;

(*Gerät 4 (CX5130-0121-M310), BOX 16*)
(*DP/DP-Kopppler*)
(*DP_State*)
	R1_B16_PB_Zustand						AT %I*: USINT;
(*Daten*)
	R1_B16_StatusModule_I_Byte_1			AT %I*: USINT;
	R1_B16_StatusModule_I_Byte_2			AT %I*: USINT;
	R1_B16_StatusModule_I_Byte_5			AT %I*: USINT;
	R1_B16_StatusModule_I_Byte_6			AT %I*: USINT;
	R1_B16_ControlModule_O					AT %Q* :ARRAY [0..4] OF USINT;
	R1_B16_VolumeFlow_I						AT %I* :UDINT;
	R1_B16_PumpLiquidTemp_I					AT %I* :UDINT;
	R1_B16_OperationTime_I					AT %I* :UDINT;
	R1_B16_ActualSetpoint_I					AT %I* :UDINT;
	R1_B16_Frequency_I						AT %I* :UDINT;
	R1_B16_UserSetpoint_I					AT %I* :UDINT;
	R1_B16_DiffPressure_I					AT %I* :UDINT;
	R1_B16_RemoteTemp2						AT %I* :UDINT;
	R1_B16_HeatEnergyCounter_I				AT %I* :UDINT;
	R1_B16_HeatDiffTemp						AT %I* :UDINT;
	R1_B16_HeatPower						AT %I* :UDINT;(* B0_SequenceNumber(1),B1AddressGenib(30),B2Class(11),B3Operation_Lenght(1),B4Data1(ID.34),Data(B5-B8) *)
	R1_B16_DirectDataReques_Temp_Geni		AT %Q* :PB_GenibusType;
	R1_B16_DirectDataReply_Temp_Geni		AT %I* :PB_GenibusType;


	R1_B16_NumberOfStarts					AT %I*	: 	UDINT;
	R1_B16_ActualSetpoint					AT %I*	:	UDINT;
	R1_B16_OperationTime					AT %I*	: 	UDINT;
	R1_B16_Speed							AT %I*	:	UDINT;
	R1_B16_Energy							AT %I*	: 	UDINT;
	R1_B16_Power							AT %I*	:	UDINT;
	R1_B16_PowerElectronicsTemp				AT %I*	:	UDINT;
	R1_B16_FaultCode						AT %I*	:	USINT;
	R1_B16_Volume							AT %I*	:	UDINT;
	R1_B16_WarningCode						AT %I*	:	USINT;

(*Gerät 4 (CX5130-0121-M310), BOX 17*)
(*DP/DP-Kopppler*)
(*DP_State*)
	R1_B17_PB_Zustand						AT %I*: USINT;
(*Daten*)
	R1_B17_StatusModule_I_Byte_1			AT %I*: USINT;
	R1_B17_StatusModule_I_Byte_2			AT %I*: USINT;
	R1_B17_StatusModule_I_Byte_5			AT %I*: USINT;
	R1_B17_StatusModule_I_Byte_6			AT %I*: USINT;
	R1_B17_ControlModule_O					AT %Q* :ARRAY [0..4] OF USINT;
	R1_B17_VolumeFlow_I						AT %I* :UDINT;
	R1_B17_PumpLiquidTemp_I					AT %I* :UDINT;
	R1_B17_OperationTime_I					AT %I* :UDINT;
	R1_B17_ActualSetpoint_I					AT %I* :UDINT;
	R1_B17_Frequency_I						AT %I* :UDINT;
	R1_B17_UserSetpoint_I					AT %I* :UDINT;
	R1_B17_DiffPressure_I					AT %I* :UDINT;
	R1_B17_RemoteTemp2						AT %I* :UDINT;
	R1_B17_HeatEnergyCounter_I				AT %I* :UDINT;
	R1_B17_HeatDiffTemp						AT %I* :UDINT;
	R1_B17_HeatPower						AT %I* :UDINT;(* B0_SequenceNumber(1),B1AddressGenib(30),B2Class(11),B3Operation_Lenght(1),B4Data1(ID.34),Data(B5-B8) *)
	R1_B17_DirectDataReques_Temp_Geni		AT %Q* :PB_GenibusType;
	R1_B17_DirectDataReply_Temp_Geni		AT %I* :PB_GenibusType;


	R1_B17_NumberOfStarts					AT %I*	: 	UDINT;
	R1_B17_ActualSetpoint					AT %I*	:	UDINT;
	R1_B17_OperationTime					AT %I*	: 	UDINT;
	R1_B17_Speed							AT %I*	:	UDINT;
	R1_B17_Energy							AT %I*	: 	UDINT;
	R1_B17_Power							AT %I*	:	UDINT;
	R1_B17_PowerElectronicsTemp				AT %I*	:	UDINT;
	R1_B17_FaultCode						AT %I*	:	USINT;
	R1_B17_Volume							AT %I*	:	UDINT;
	R1_B17_WarningCode						AT %I*	:	USINT;

(*Gerät 4 (CX5130-0121-M310), BOX 18*)
(*DP/DP-Kopppler*)
		(* Variablen in Globale Variablen   AC_PB_Var definiert
		Anbindung Atlas Copco MK5 Profibus Gateway Compressor *)


(* Janitza UMG 604 in Druckluftkompressor*)
	R1_B19_Request							AT %Q* 	:	BYTE;
	R1_B19_In								AT %I*	:	ARRAY[0..31] OF UINT;


(*Master*)
(*Gerät 6 (EL6731), BOX 01*)
(*DP/DP-Kopppler*)
(*DP_State*)
	R2_B01_PB_Zustand						AT %I*: USINT;
(*Daten*)
	R2_B01_StatusModule_I_Byte_1			AT %I*: USINT;
	R2_B01_StatusModule_I_Byte_2			AT %I*: USINT;
	R2_B01_StatusModule_I_Byte_5			AT %I*: USINT;
	R2_B01_StatusModule_I_Byte_6			AT %I*: USINT;
	R2_B01_ControlModule_O					AT %Q* :ARRAY [0..4] OF USINT;  (*Control Modul muss getestet werden*)
	R2_B01_VolumeFlow_I						AT %I* :UDINT;
	R2_B01_PumpLiquidTemp_I					AT %I* :UDINT;
	R2_B01_OperationTime_I					AT %I* :UDINT;
	R2_B01_ActualSetpoint_I					AT %I* :UDINT;
	R2_B01_Frequency_I						AT %I* :UDINT;
	R2_B01_UserSetpoint_I					AT %I* :UDINT;
	R2_B01_DiffPressure_I					AT %I* :UDINT;
	R2_B01_RemoteTemp2						AT %I* :UDINT;
	R2_B01_HeatEnergyCounter_I				AT %I* :UDINT;
	R2_B01_HeatDiffTemp						AT %I* :UDINT;
	R2_B01_HeatPower						AT %I* :UDINT;(* B0_SequenceNumber(1),B1AddressGenib(30),B2Class(11),B3Operation_Lenght(1),B4Data1(ID.34),Data(B5-B8) *)
	R2_B01_DirectDataReques_Temp_Geni		AT %Q* :PB_GenibusType;
	R2_B01_DirectDataReply_Temp_Geni		AT %I* :PB_GenibusType;

	R2_B01_NumberOfStarts					AT %I*	: 	UDINT;
	R2_B01_ActualSetpoint					AT %I*	:	UDINT;
	R2_B01_OperationTime					AT %I*	: 	UDINT;
	R2_B01_Speed							AT %I*	:	UDINT;
	R2_B01_Energy							AT %I*	: 	UDINT;
	R2_B01_Power							AT %I*	:	UDINT;
	R2_B01_PowerElectronicsTemp				AT %I*	:	UDINT;
	R2_B01_FaultCode						AT %I*	:	USINT;
	R2_B01_Volume							AT %I*	:	UDINT;
	R2_B01_WarningCode						AT %I*	:	USINT;


(*Gerät 6 (EL6731), BOX 02*)
(*DP/DP-Kopppler*)
(*DP_State*)
	R2_B02_PB_Zustand						AT %I*: USINT;
(*Daten*)
	R2_B02_StatusModule_I_Byte_1			AT %I*: USINT;
	R2_B02_StatusModule_I_Byte_2			AT %I*: USINT;
	R2_B02_StatusModule_I_Byte_5			AT %I*: USINT;
	R2_B02_StatusModule_I_Byte_6			AT %I*: USINT;
	R2_B02_ControlModule_O					AT %Q* :ARRAY [0..4] OF USINT;
	R2_B02_VolumeFlow_I						AT %I* :UDINT;
	R2_B02_PumpLiquidTemp_I					AT %I* :UDINT;
	R2_B02_OperationTime_I					AT %I* :UDINT;
	R2_B02_ActualSetpoint_I					AT %I* :UDINT;
	R2_B02_Frequency_I						AT %I* :UDINT;
	R2_B02_UserSetpoint_I					AT %I* :UDINT;
	R2_B02_DiffPressure_I					AT %I* :UDINT;
	R2_B02_RemoteTemp2						AT %I* :UDINT;
	R2_B02_HeatEnergyCounter_I				AT %I* :UDINT;
	R2_B02_HeatDiffTemp						AT %I* :UDINT;
	R2_B02_HeatPower						AT %I* :UDINT;(* B0_SequenceNumber(1),B1AddressGenib(30),B2Class(11),B3Operation_Lenght(1),B4Data1(ID.34),Data(B5-B8) *)
	R2_B02_DirectDataReques_Temp_Geni		AT %Q* :PB_GenibusType;
	R2_B02_DirectDataReply_Temp_Geni		AT %I* :PB_GenibusType;

	R2_B02_NumberOfStarts					AT %I*	: 	UDINT;
	R2_B02_ActualSetpoint					AT %I*	:	UDINT;
	R2_B02_OperationTime					AT %I*	: 	UDINT;
	R2_B02_Speed							AT %I*	:	UDINT;
	R2_B02_Energy							AT %I*	: 	UDINT;
	R2_B02_Power							AT %I*	:	UDINT;
	R2_B02_PowerElectronicsTemp				AT %I*	:	UDINT;
	R2_B02_FaultCode						AT %I*	:	USINT;
	R2_B02_Volume							AT %I*	:	UDINT;
	R2_B02_WarningCode						AT %I*	:	USINT;


(*Gerät 6 (EL6731), BOX 03*)
(*DP/DP-Kopppler*)
(*DP_State*)
	R2_B03_PB_Zustand						AT %I*: USINT;
(*Daten*)
	R2_B03_StatusModule_I_Byte_1			AT %I*: USINT;
	R2_B03_StatusModule_I_Byte_2			AT %I*: USINT;
	R2_B03_StatusModule_I_Byte_5			AT %I*: USINT;
	R2_B03_StatusModule_I_Byte_6			AT %I*: USINT;
	R2_B03_ControlModule_O					AT %Q* :ARRAY [0..4] OF USINT;
	R2_B03_VolumeFlow_I						AT %I* :UDINT;
	R2_B03_PumpLiquidTemp_I					AT %I* :UDINT;
	R2_B03_OperationTime_I					AT %I* :UDINT;
	R2_B03_ActualSetpoint_I					AT %I* :UDINT;
	R2_B03_Frequency_I						AT %I* :UDINT;
	R2_B03_UserSetpoint_I					AT %I* :UDINT;
	R2_B03_DiffPressure_I					AT %I* :UDINT;
	R2_B03_RemoteTemp2						AT %I* :UDINT;
	R2_B03_HeatEnergyCounter_I				AT %I* :UDINT;
	R2_B03_HeatDiffTemp						AT %I* :UDINT;
	R2_B03_HeatPower						AT %I* :UDINT;(* B0_SequenceNumber(1),B1AddressGenib(30),B2Class(11),B3Operation_Lenght(1),B4Data1(ID.34),Data(B5-B8) *)
	R2_B03_DirectDataReques_Temp_Geni		AT %Q* :PB_GenibusType;
	R2_B03_DirectDataReply_Temp_Geni		AT %I* :PB_GenibusType;

	R2_B03_NumberOfStarts					AT %I*	: 	UDINT;
	R2_B03_ActualSetpoint					AT %I*	:	UDINT;
	R2_B03_OperationTime					AT %I*	: 	UDINT;
	R2_B03_Speed							AT %I*	:	UDINT;
	R2_B03_Energy							AT %I*	: 	UDINT;
	R2_B03_Power							AT %I*	:	UDINT;
	R2_B03_PowerElectronicsTemp				AT %I*	:	UDINT;
	R2_B03_FaultCode						AT %I*	:	USINT;
	R2_B03_Volume							AT %I*	:	UDINT;
	R2_B03_WarningCode						AT %I*	:	USINT;


(*Gerät 6 (EL6731), BOX 04*)
(*DP/DP-Kopppler*)
(*DP_State*)
	R2_B04_PB_Zustand						AT %I*: USINT;
(*Daten*)
	R2_B04_StatusModule_I_Byte_1			AT %I*: USINT;
	R2_B04_StatusModule_I_Byte_2			AT %I*: USINT;
	R2_B04_StatusModule_I_Byte_5			AT %I*: USINT;
	R2_B04_StatusModule_I_Byte_6				AT %I*	:	 USINT;
	R2_B04_ControlModule_O					AT %Q* 	:	ARRAY [0..4] OF USINT;
	R2_B04_VolumeFlow_I						AT %I* 	:	UDINT;
	R2_B04_PumpLiquidTemp_I				AT %I* 	:	UDINT;
	R2_B04_OperationTime_I					AT %I* 	:	UDINT;
	R2_B04_ActualSetpoint_I					AT %I* 	:	UDINT;
	R2_B04_Frequency_I						AT %I* 	:	UDINT;
	R2_B04_UserSetpoint_I					AT %I* 	:	UDINT;
	R2_B04_DiffPressure_I						AT %I* 	:	UDINT;
	R2_B04_RemoteTemp2					AT %I* 	:	UDINT;
	R2_B04_HeatEnergyCounter_I				AT %I* 	:	UDINT;
	R2_B04_HeatDiffTemp						AT %I* 	:	UDINT;
	R2_B04_HeatPower						AT %I* 	:	UDINT;(* B0_SequenceNumber(1),B1AddressGenib(30),B2Class(11),B3Operation_Lenght(1),B4Data1(ID.34),Data(B5-B8) *)
	R2_B04_DirectDataReques_Temp_Geni		AT %Q* 	:	PB_GenibusType;
	R2_B04_DirectDataReply_Temp_Geni		AT %I* 	:	PB_GenibusType;

	R2_B04_NumberOfStarts					AT %I*	: 	UDINT;
	R2_B04_ActualSetpoint					AT %I*	:	UDINT;
	R2_B04_OperationTime					AT %I*	: 	UDINT;
	R2_B04_Speed							AT %I*	:	UDINT;
	R2_B04_Energy							AT %I*	: 	UDINT;
	R2_B04_Power							AT %I*	:	UDINT;
	R2_B04_PowerElectronicsTemp				AT %I*	:	UDINT;
	R2_B04_FaultCode						AT %I*	:	USINT;
	R2_B04_Volume							AT %I*	:	UDINT;
	R2_B04_WarningCode						AT %I*	:	USINT;


(*Gerät 6 (EL6731), BOX 05*)
(*DP/DP-Kopppler*)
(*DP_State*)
	R2_B05_PB_Zustand						AT %I*: USINT;
(*Daten*)
	R2_B05_StatusModule_I_Byte_1			AT %I*: USINT;
	R2_B05_StatusModule_I_Byte_2			AT %I*: USINT;
	R2_B05_StatusModule_I_Byte_5			AT %I*: USINT;
	R2_B05_StatusModule_I_Byte_6			AT %I*: USINT;
	R2_B05_ControlModule_O					AT %Q* :ARRAY [0..4] OF USINT;
	R2_B05_VolumeFlow_I						AT %I* :UDINT;
	R2_B05_PumpLiquidTemp_I					AT %I* :UDINT;
	R2_B05_OperationTime_I					AT %I* :UDINT;
	R2_B05_ActualSetpoint_I					AT %I* :UDINT;
	R2_B05_Frequency_I						AT %I* :UDINT;
	R2_B05_UserSetpoint_I					AT %I* :UDINT;
	R2_B05_DiffPressure_I					AT %I* :UDINT;
	R2_B05_RemoteTemp2						AT %I* :UDINT;
	R2_B05_HeatEnergyCounter_I				AT %I* :UDINT;
	R2_B05_HeatDiffTemp						AT %I* :UDINT;
	R2_B05_HeatPower						AT %I* :UDINT;(* B0_SequenceNumber(1),B1AddressGenib(30),B2Class(11),B3Operation_Lenght(1),B4Data1(ID.34),Data(B5-B8) *)
	R2_B05_DirectDataReques_Temp_Geni		AT %Q* :PB_GenibusType;
	R2_B05_DirectDataReply_Temp_Geni		AT %I* :PB_GenibusType;

	R2_B05_NumberOfStarts					AT %I*	: 	UDINT;
	R2_B05_ActualSetpoint					AT %I*	:	UDINT;
	R2_B05_OperationTime					AT %I*	: 	UDINT;
	R2_B05_Speed							AT %I*	:	UDINT;
	R2_B05_Energy							AT %I*	: 	UDINT;
	R2_B05_Power							AT %I*	:	UDINT;
	R2_B05_PowerElectronicsTemp				AT %I*	:	UDINT;
	R2_B05_FaultCode						AT %I*	:	USINT;
	R2_B05_Volume							AT %I*	:	UDINT;
	R2_B05_WarningCode						AT %I*	:	USINT;


(*Gerät 6 (EL6731), BOX 06*)
(*DP/DP-Kopppler*)
(*DP_State*)
	R2_B06_PB_Zustand						AT %I*: USINT;
(*Daten*)
	R2_B06_StatusModule_I_Byte_1			AT %I*: USINT;
	R2_B06_StatusModule_I_Byte_2			AT %I*: USINT;
	R2_B06_StatusModule_I_Byte_5			AT %I*: USINT;
	R2_B06_StatusModule_I_Byte_6			AT %I*: USINT;
	R2_B06_ControlModule_O					AT %Q* :ARRAY [0..4] OF USINT;
	R2_B06_VolumeFlow_I						AT %I* :UDINT;
	R2_B06_PumpLiquidTemp_I					AT %I* :UDINT;
	R2_B06_OperationTime_I					AT %I* :UDINT;
	R2_B06_ActualSetpoint_I					AT %I* :UDINT;
	R2_B06_Frequency_I						AT %I* :UDINT;
	R2_B06_UserSetpoint_I					AT %I* :UDINT;
	R2_B06_DiffPressure_I					AT %I* :UDINT;
	R2_B06_RemoteTemp2						AT %I* :UDINT;
	R2_B06_HeatEnergyCounter_I				AT %I* :UDINT;
	R2_B06_HeatDiffTemp						AT %I* :UDINT;
	R2_B06_HeatPower						AT %I* :UDINT;(* B0_SequenceNumber(1),B1AddressGenib(30),B2Class(11),B3Operation_Lenght(1),B4Data1(ID.34),Data(B5-B8) *)
	R2_B06_DirectDataReques_Temp_Geni		AT %Q* :PB_GenibusType;
	R2_B06_DirectDataReply_Temp_Geni		AT %I* :PB_GenibusType;

	R2_B06_NumberOfStarts					AT %I*	: 	UDINT;
	R2_B06_ActualSetpoint					AT %I*	:	UDINT;
	R2_B06_OperationTime					AT %I*	: 	UDINT;
	R2_B06_Speed							AT %I*	:	UDINT;
	R2_B06_Energy							AT %I*	: 	UDINT;
	R2_B06_Power							AT %I*	:	UDINT;
	R2_B06_PowerElectronicsTemp				AT %I*	:	UDINT;
	R2_B06_FaultCode						AT %I*	:	USINT;
	R2_B06_Volume							AT %I*	:	UDINT;
	R2_B06_WarningCode						AT %I*	:	USINT;

*)

END_VAR

// ---- Global Variables/Global_Variables.TcGVL
{attribute 'Tc2GvlVarNames'}
VAR_GLOBAL
	GA_Allgemein 	: FB_GA_Allgemein;
	{attribute 'OPC.UA.DA' := '1'} GA_global		: ST_GA_global;		

	(* Kategorien Programme *)
	Wetterstation				: FB_WS;
	Heizung_Lueftung_Klima		: FB_HLK;
	Wandler						: FB_WDL;
	Speicher					: FB_SPR;
	Netze						: FB_NTZ;
	Umwelt						: FB_UMWELT;
	Management					: FB_MGMT;

	Beleuchtung					: FB_Beleuchtung;

	Anlagenversorgung			: FB_AV;
	Zaehler						: FB_ZAE;
	Signal_Ampel				: FB_System_Ampel;
	Counter_Genibus				: DINT;

	Dali_K522A1_DALI_IN		 	AT %I* : ST_DALIV2InData;	(*~ Eingangspuffer für Dali Klemme *)
	Dali_K522A1_DALI_OUT 		AT %Q* : ST_DALIV2OutData;	(*~ Ausgangspuffer für Dali Klemme *)

	(* Wetterstation *)
	KL_Wetterstation			: KL6301;
	KL_Wetterstation_IN			AT %I* : ARRAY[1..24]OF BYTE;
	KL_Wetterstation_OUT		AT %Q* : ARRAY[1..24]OF BYTE;

	Initialisierung				: ST_Initialisierungsroutine;
	Initialisierungsroutine	: FB_Initialisierungsroutine;

END_VAR

// ---- POUs/com_task.TcPOU
PROGRAM com_task
VAR
	try : BOOL := FALSE;
END_VAR

(* Zähler *)
Zaehler();

(* Wetterstation *)
Wetterstation();


try :=  TRUE;

END_PROGRAM

// ---- POUs/Umwelt/FB_UMWELT.TcPOU
FUNCTION_BLOCK FB_UMWELT
VAR_INPUT
END_VAR
VAR_OUTPUT
END_VAR
VAR

	(*TF_aussen				: FB_TF;*)

	{attribute 'OPC.UA.DA' := '1'}Daemmerung				: REAL;
	{attribute 'OPC.UA.DA' := '1'}Temp_Aussen_WS_Mittelw	: REAL;
	{attribute 'OPC.UA.DA' := '1'}Temp_Aussen_WS			: REAL;
	{attribute 'OPC.UA.DA' := '1'}Regen					: BOOL;		
	{attribute 'OPC.UA.DA' := '1'}Windgeschwindigkeit		: REAL;

	(* Mittelwert	berechnung	: FB_CTRL_MOVING_AVERAGE;	*)

	{attribute 'OPC.UA.DA' := '1'}Temp_Aussen			: REAL;		
	{attribute 'OPC.UA.DA' := '1'}Temp_Aussen_Mittelw	: REAL;		
	{attribute 'OPC.UA.DA' := '1'}Temp_Halle_Sektor1		: REAL;	
	{attribute 'OPC.UA.DA' := '1'}Temp_Halle_Sektor2		: REAL;	
	{attribute 'OPC.UA.DA' := '1'}Temp_Halle_Sektor3		: REAL;	

	Tempfuehler_Halle_Sektor1				: FB_TF;
	Tempfuehler_Halle_Sektor2				: FB_TF;
	Tempfuehler_Halle_Sektor3				: FB_TF;
	Tempfuehler_Temperatur_Aussen_TF		: FB_TF;

	Tagesmittelung							: FB_UW_Temp_Mittelung;

END_VAR

Temp_Aussen_WS := Wetterstation.Wetterstation_Lesen.Aussentemperatur;
Temp_Aussen_WS_Mittelw := Wetterstation.Wetterstation_Lesen.Aussentemperatur_gemittelt;
Daemmerung := Wetterstation.Wetterstation_Lesen.Daemmerung;
Regen := Wetterstation.Wetterstation_Lesen.Regensensor;
Windgeschwindigkeit := Wetterstation.Wetterstation_Lesen.Windgeschwindigkeit;
Temp_Aussen := Wetterstation.Wetterstation_Lesen.Aussentemperatur;
Temp_Halle_Sektor1 := Tempfuehler_Halle_Sektor1.Temperatur;
Temp_Halle_Sektor2 := Tempfuehler_Halle_Sektor2.Temperatur;
Temp_Halle_Sektor3 := Tempfuehler_Halle_Sektor3.Temperatur;
// 16.10.19: Wetterstation kaputt, deswegen 12 Grad als Standardwert. Rücksetzen, wenn sie wieder funktioniert.
Tempfuehler_Halle_Sektor1(); // FB_TF
Tempfuehler_Halle_Sektor2(); // FB_TF
Tempfuehler_Halle_Sektor3(); // FB_TF
Tempfuehler_Temperatur_Aussen_TF(); // FB_TF
Temp_Aussen_Mittelw := Wetterstation.Wetterstation_Lesen.Aussentemperatur_gemittelt;
Tagesmittelung(Einzelwert := Tempfuehler_Temperatur_Aussen_TF.Temperatur); // FB_UW_Temp_Mittelung
// Wetterstation.Wetterstation_Lesen.Aussentemperatur: input not connected

END_FUNCTION_BLOCK

// ---- POUs/Management/FB_MGMT.TcPOU
FUNCTION_BLOCK FB_MGMT
VAR_INPUT
	Freigabe_auto			: BOOL;
	Freigabe_Deakt_auto		: BOOL;
	Betrieb_Anford_auto		: BOOL;
	Regelung_Modus_auto		: SINT;
	Regelung_Sollw_auto		: REAL;
END_VAR
VAR_OUTPUT
END_VAR
VAR
	Netze_MGMT		    	: FB_MGMT_ThNTZ;
	Betonspeicher			: FB_MGMT_BSp;

	{attribute 'OPC.UA.DA' := '1'}Steuerung				: ST_FB_MGMT_Steuerung;		
	{attribute 'OPC.UA.DA' := '1'}Stellwert				: ST_FB_MGMT_Stellwert;		
	{attribute 'OPC.UA.DA' := '1'}Zustand					: ST_FB_MGMT_Zustand;	
	{attribute 'OPC.UA.DA' := '1'}Parameter				: ST_FB_MGMT_Parameter;		

    Zustandscheck			: FB_MGMT_Zustandscheck;
	Logik					: FB_MGMT_Logik;
	Ablaufsteuerung			: FB_MGMT_Ablaufsteuerung;
	Sollwertscheck			: FB_MGMT_Sollwertscheck;
	Regelung				: FB_MGMT_Regelung;
	Zuweisungen				: FB_Zuweisungen;

END_VAR

Netze_MGMT(); // FB_MGMT_ThNTZ
Parameter := Initialisierung.MGMT_Parameter;
Steuerung.Freigabe.auto := Freigabe_auto;
Steuerung.Freigabe_Deakt.auto := Freigabe_Deakt_auto;
Steuerung.Betrieb_Anford.auto := Betrieb_Anford_auto;
Steuerung.Regelung_Modus.auto := Regelung_Modus_auto;
Steuerung.Regelung_Sollw.auto := Regelung_Sollw_auto;
Zuweisungen(Zustand := Zustand); // FB_Zuweisungen
Betonspeicher(
    Parameter := Parameter,
    Zustand_BSp_WW := Speicher.System_Betonspeicher_Warmwasser_797.Betonspeicher_797.Zustand,
    Zustand_BSp_KW := Speicher.System_Betonspeicher_Kaltwasser_795.Betonspeicher_795.Zustand,
    Zustand_System_AFA := Wandler.System_Aussenfassadenaktivierung_600.Zustand,
    Stellwert := Stellwert,
    Zustand := Zustand); // FB_MGMT_BSp
Zustandscheck(Parameter := Parameter, Steuerung := Steuerung, Zustand := Zustand); // FB_MGMT_Zustandscheck
Logik(Parameter := Parameter, Steuerung := Steuerung, Zustand := Zustand); // FB_MGMT_Logik
Ablaufsteuerung(Zustand := Zustand, Stellwert := Stellwert, Steuerung := Steuerung); // FB_MGMT_Ablaufsteuerung
Sollwertscheck(Steuerung := Steuerung, Parameter := Parameter, Zustand := Zustand); // FB_MGMT_Sollwertscheck
Regelung(Steuerung := Steuerung, Parameter := Parameter, Stellwert := Stellwert, Zustand := Zustand); // FB_MGMT_Regelung

END_FUNCTION_BLOCK

// ---- POUs/Management/Alte Struktur/FB_MGMT_ThNTZ.TcPOU
FUNCTION_BLOCK FB_MGMT_ThNTZ
VAR_INPUT
END_VAR
VAR_OUTPUT
END_VAR
VAR
	System_Waermetauscher_915				: FB_MGMT_ThNTZ_Aktor;
END_VAR

System_Waermetauscher_915(
    Stellwert_Netz_KW := Netze.Kaltwasser_1xx.Stellwert,
    Stellwert_Netz_WW := Netze.Warmwasser_2xx.Stellwert,
    Stellwert_Netz_HW := Netze.Heisswasser_3xx.Stellwert,
    Aktor_Netze_Anford := Wandler.System_Waermetauscher_915.Zustand.Netze_Anford,
    Zustand_Netz_KW := Netze.Kaltwasser_1xx.Zustand,
    Zustand_Netz_WW := Netze.Warmwasser_2xx.Zustand,
    Zustand_Netz_HW := Netze.Heisswasser_3xx.Zustand); // FB_MGMT_ThNTZ_Aktor

END_FUNCTION_BLOCK

// ---- POUs/Management/Alte Struktur/FB_MGMT_ThNTZ_Aktor.TcPOU
FUNCTION_BLOCK FB_MGMT_ThNTZ_Aktor
VAR_IN_OUT
	Zustand_Netz_KW		: ST_ThNTZ_Zustand;
	Zustand_Netz_WW	: ST_ThNTZ_Zustand;
	Zustand_Netz_HW	: ST_ThNTZ_Zustand;
END_VAR
VAR_INPUT
	Stellwert_Netz_KW	: ST_ThNTZ_Stellwert;
	Stellwert_Netz_WW	: ST_ThNTZ_Stellwert;
	Stellwert_Netz_HW	: ST_ThNTZ_Stellwert;

	Aktor_Netze_Anford	: ST_Zustand_Netze_Anford;
END_VAR
VAR_OUTPUT
	{attribute 'OPC.UA.DA' := '1'}Stellwert		: ST_MGMT_ThNTZ_Aktor_Stellwert;	
	{attribute 'OPC.UA.DA' := '1'}Parameter	: ST_MGMT_ThNTZ_Aktor_Parameter;		
	Zustand		: ST_MGMT_ThNTZ_Aktor_Zustand;
END_VAR
VAR
	Hysterese_KW_Heizung			: FB_CTRL_2POINT;
	Hysterese_KW_Kuehlung			: FB_CTRL_2POINT;
	Hysterese_WW_Heizung			: FB_CTRL_2POINT;
	Hysterese_WW_Kuehlung			: FB_CTRL_2POINT;
	Hysterese_HW_Heizung			: FB_CTRL_2POINT;
	Hysterese_HW_Kuehlung			: FB_CTRL_2POINT;
	Hysterese_Parameter				: ST_CTRL_2POINT_PARAMS;
END_VAR

